	    // trigger kaxon horn: rising trigger of start
	    #RT_Start(CLK := #Start);
	    // trigger kaxon horn: rising trigger of stop
	    #RT_Stop(CLK := #Stop);
	    // trigger kaxon horn: rising trigger of fault
	    #RT_Fault(CLK := #GlobalFault);
	    // trigger kaxon horn: rising trigger of blockage
	    #RT_Blockage(CLK := #GlobalBlockage);
	    // trigger kaxon horn: rising trigger of estop
	    #RT_Estop(CLK := #EstopActive);
	    // trigger kaxon horn: rising trigger of fire
	    #RT_Fire(CLK := #Fire);
	    
	    // --------------
	    // Horn condition
	    // --------------
	    
	    #HornCondition :=
	    #RT_Start.Q OR
	    #RT_Stop.Q OR
	    #RT_Fire.Q OR
	    #RT_Fault.Q OR
	    #RT_Estop.Q OR
	    #RT_Fire.Q;
	    
	    // -------------------
	    // Horn alert duration
	    // -------------------
	    
	    #KlaxonHornTimer.TOF(IN := #HornCondition,
	                         PT := t#5s);
	    
	    #HornActive :=
	    #KlaxonHornTimer.Q;
	    
	END_REGION
	
	
	
	
	
	
	
	
	
	
	
	
	
END_FUNCTION_BLOCK
END_NAMESPACE

NAMESPACE ProductionLine
FUNCTION_BLOCK Flow_Test
{ S7_Optimized_Access := 'TRUE' ; Published := 'FALSE' }
VERSION : 0.1
   VAR 
      Start { S7_SetPoint := 'True'} : Bool;   //  // Start command (e.g. from I0.0)
      StartTest : Test_Logic;
      GoToRightDP1 : Test_Logic;
      ContinueStraightDP1 : Test_Logic;
      ContinueStraightDP2 : Test_Logic;
      GotorightDP2Thentoright : Test_Logic;
      GotorightDP2ThentoLeft : Test_Logic;
      ContinueStraightDP3 : Test_Logic;
      ContinueStraightDP4 : Test_Logic;
      GotoRightDP4 : Test_Logic;
      "A1.13.1_Straight" : Test_Logic;
      "A1.13.1_left" : Test_Logic;
      R_TRIG_Instance {InstructionName := 'R_TRIG'; LibVersion := '1.0'} : R_TRIG;
   END_VAR


BEGIN
	// ==========================================================================================================================================
	// Company        : LogTech, s.r.o.
	// Created by     : Mahmoud Elnady
	// Block          : FB_FlowTest
	// Project        : Lékárna Chrudim
	// Project number : 23-157
	// ==========================================================================================================================================
	
	REGION Start Test
	    #StartTest(Start := #Start,
	               StartPoint := _."A1.1.1",
	               EndPoint :=  _."A1.5.3");
	END_REGION
	
	
	REGION Go TO Right DP1
	    #GoToRightDP1(Start := DB_ToteTracking.Conveyor[_."A1.6.1"].ToteDir.toRight AND
	                  DB_ToteTracking.Conveyor[_."A1.6.2"].ToteDir.toRight AND
	                  _.ProductionLine.IDB_ProductionLine."A1.5.3".FilteredSensor,
	                  StartPoint := _."B1.1.1",
	                  EndPoint := _."B1.9.2");
	END_REGION
	
	
	REGION CONTINUE Straight DP1
	    
	    #ContinueStraightDP1(Start := DB_ToteTracking.Conveyor[_."A1.6.1"].ToteDir.Straight AND
	                         DB_ToteTracking.Conveyor[_."A1.6.2"].ToteDir.Straight AND
	                         _.ProductionLine.IDB_ProductionLine."A1.5.3".FilteredSensor,
	                         StartPoint := _."A1.7.1",
	                         EndPoint := _."A1.8.1");
	    
	END_REGION
	
	IF (DB_ToteTracking.Conveyor[_."A1.6.1"].ToteDir.Straight OR
	    DB_ToteTracking.Conveyor[_."A1.6.1"].ToteDir.toRight) AND
	    IDB_ProductionLine."A1.5.3".FilteredSensor
	THEN
	    _.Global.DB_SystemSimu.TriggerSensor.Line.ProductionLine.Conveyor[_."A1.6.1"] := TRUE;
	ELSE
	    _.Global.DB_SystemSimu.TriggerSensor.Line.ProductionLine.Conveyor[_."A1.6.1"] := FALSE;
	END_IF;
	
	
	        
	REGION CONTINUE Straight DP2
	    
	    #ContinueStraightDP2(Start := DB_ToteTracking.Conveyor[_."B1.10.1"].ToteDir.Straight AND
	                                  IDB_ProductionLine."B1.9.2".FilteredSensor,
	                         StartPoint := _."B1.11.1",
	                         EndPoint := _."B1.17.4");
	    
	END_REGION
	
	
	REGION Go TO Right DP2 THEN TO Right
	    #GotorightDP2Thentoright(Start := DB_ToteTracking.Conveyor[_."B1.10.1"].ToteDir.toRight AND
	                             DB_ToteTracking.Conveyor[_."C1.3.1"].ToteDir.toRight AND
	                             IDB_ProductionLine."B1.9.2".FilteredSensor,
	                             StartPoint := _."C1.2.2",
	                             EndPoint := _."C1.2.1");
	END_REGION
	
	
	REGION Go TO Right THEN TO Left
	    #GotorightDP2ThentoLeft(Start := DB_ToteTracking.Conveyor[_."B1.10.1"].ToteDir.toRight AND
	                            DB_ToteTracking.Conveyor[_."C1.3.1"].ToteDir.toLeft AND
	                            IDB_ProductionLine."B1.9.2".FilteredSensor,
	                            StartPoint := _."C1.4.1",
	                            EndPoint :=  _."C1.4.2");
	END_REGION
	
	
	IF (DB_ToteTracking.Conveyor[_."B1.10.1"].ToteDir.Straight OR
	    DB_ToteTracking.Conveyor[_."B1.10.1"].ToteDir.toRight) AND
	    IDB_ProductionLine."B1.9.2".FilteredSensor
	THEN
	    _.Global.DB_SystemSimu.TriggerSensor.Line.ProductionLine.Conveyor[_."B1.10.1"] := TRUE;
	ELSE
	    _.Global.DB_SystemSimu.TriggerSensor.Line.ProductionLine.Conveyor[_."B1.10.1"] := FALSE;
	END_IF;
	
	IF (DB_ToteTracking.Conveyor[_."C1.3.1"].ToteDir.toLeft OR
	    DB_ToteTracking.Conveyor[_."C1.3.1"].ToteDir.toRight) AND
	    IDB_ProductionLine."B1.10.1".FilteredSensor AND
	    DB_ToteTracking.Conveyor[_."B1.10.1"].ToteDir.toRight
	THEN
	    _.Global.DB_SystemSimu.TriggerSensor.Line.ProductionLine.Conveyor[_."C1.3.1"] := TRUE;
	ELSE
	    _.Global.DB_SystemSimu.TriggerSensor.Line.ProductionLine.Conveyor[_."C1.3.1"] := FALSE;
	END_IF;
	
	
	
	REGION CONTINUE Straight DP3
	    #ContinueStraightDP3(Start := DB_ToteTracking.Conveyor[_."B1.18.1"].ToteDir.Straight AND
	                                  IDB_ProductionLine."B1.17.4".FilteredSensor,
	                         StartPoint := _."B1.19.1",
	                         EndPoint := _."B1.23.1");
	END_REGION
	
	IF (DB_ToteTracking.Conveyor[_."B1.18.1"].ToteDir.toLeft OR
	    DB_ToteTracking.Conveyor[_."B1.18.1"].ToteDir.Straight) AND
	    IDB_ProductionLine."B1.17.4".FilteredSensor
	THEN
	    _.Global.DB_SystemSimu.TriggerSensor.Line.ProductionLine.Conveyor[_."B1.18.1"] := TRUE;
	ELSE
	    _.Global.DB_SystemSimu.TriggerSensor.Line.ProductionLine.Conveyor[_."B1.18.1"] := FALSE;
	END_IF;
	
	#R_TRIG_Instance(CLK:=( IDB_ProductionLine."B1.18.1".FilteredSensor AND
	                 DB_ToteTracking.Conveyor[_."B1.18.1"].ToteDir.toLeft));
	
	
	
	REGION CONTINUE Straight DP4
	    #ContinueStraightDP4(Start := DB_ToteTracking.Conveyor[_."A1.9.1"].ToteDir.Straight AND
	                         DB_ToteTracking.Conveyor[_."A1.9.2"].ToteDir.Straight AND
	                         _.ProductionLine.IDB_ProductionLine."A1.8.1".FilteredSensor,
	                         StartPoint := _."A1.10.1",
	                         EndPoint := _."A1.12.2");
	END_REGION
	
	
	REGION Go TO Right DP4
	    #GotoRightDP4(Start := DB_ToteTracking.Conveyor[_."A1.9.1"].ToteDir.toRight AND
	                  DB_ToteTracking.Conveyor[_."A1.9.2"].ToteDir.toRight AND
	                  _.ProductionLine.IDB_ProductionLine."A1.8.1".FilteredSensor,
	                  StartPoint := _."D1.1.1",
	                  EndPoint :=  _."D1.12.3");
	END_REGION
	
	IF (DB_ToteTracking.Conveyor[_."A1.9.1"].ToteDir.Straight OR
	    DB_ToteTracking.Conveyor[_."A1.9.1"].ToteDir.toRight) AND
	    IDB_ProductionLine."A1.8.1".FilteredSensor
	THEN
	    _.Global.DB_SystemSimu.TriggerSensor.Line.ProductionLine.Conveyor[_."A1.9.1"] := TRUE;
	ELSE
	    _.Global.DB_SystemSimu.TriggerSensor.Line.ProductionLine.Conveyor[_."A1.9.1"] := FALSE;
	END_IF;
	
	REGION A1.13.1_Straight
	    
	    #"A1.13.1_Straight"(Start:= DB_ToteTracking.Conveyor[_."A1.13.1"].ToteDir.Straight AND
	                                IDB_ProductionLine."A1.12.2".FilteredSensor,
	                        StartPoint:=_."A1.14.1",
	                        EndPoint:= _."A1.14.26");
	    
	   
	END_REGION
	        
	REGION A1.13.1_Left
	    
	    #"A1.13.1_left"(Start := DB_ToteTracking.Conveyor[_."A1.13.1"].ToteDir.toLeft AND
	                    IDB_ProductionLine."A1.12.2".FilteredSensor,
	                    StartPoint := _."A2.2.1",
	                    EndPoint := _."A2.2.26");
	    
	    
	END_REGION
	
	
	    
	    
	
END_FUNCTION_BLOCK
END_NAMESPACE

NAMESPACE ProductionLine
FUNCTION_BLOCK Test_Logic
{ S7_Optimized_Access := 'TRUE' ; Published := 'FALSE' }
VERSION : 0.1
   VAR_INPUT 
      Start : Bool;
      StartPoint : Int;
      EndPoint : Int;
   END_VAR

   VAR 
      Active : Bool;
      "Counter" : Int;
      PulseTimer {InstructionName := 'TON_TIME'; LibVersion := '1.0'; S7_SetPoint := 'False'} : TON_TIME;
   END_VAR


BEGIN
	// ==========================================================================================================================================
	// Company        : LogTech, s.r.o.
	// Created by     : Mahmoud Elnady
	// Block          : FB_LineA1
	// Project        : Lékárna Chrudim
	// Project number : 23-157
	// ==========================================================================================================================================
	
	REGION Start
	    // Start sequence
	    IF #Start AND NOT #Active THEN
	        #Active := TRUE;
	        #Counter := #StartPoint;               // Start from first output
	    END_IF;
	    
	    // Main pulse logic
	    IF #Active THEN
	        // Turn ON the current output
	        _.Global.DB_SystemSimu.TriggerSensor.Line.ProductionLine.Conveyor[#Counter] := TRUE;
	        #PulseTimer(IN := TRUE,
	                    PT := T#3s);
	        
	        // When timer expires
	        IF #PulseTimer.Q THEN
	            // Turn OFF current output
	            _.Global.DB_SystemSimu.TriggerSensor.Line.ProductionLine.Conveyor[#Counter] := FALSE;
	            
	            // Reset timer
	            RESET_TIMER(#PulseTimer);
	            
	            // Move to next output
	            #Counter := #Counter + 1;
	            
	            // Stop if last output finished
	            IF #Counter > #EndPoint THEN
	                #Active := FALSE;
	            END_IF;
	        END_IF;
	    ELSE
	        // Make sure all outputs are OFF when not active
	        (* FOR #var_i := 1001 TO #N DO
	        //#Q[#var_i] := FALSE;
	        _.Global.DB_SystemSimu.TriggerSensor.Line.ProductionLine.Conveyor[#Counter] := FALSE;
	    END_FOR;*)
	        RESET_TIMER(#PulseTimer);
	    END_IF;
	END_REGION
END_FUNCTION_BLOCK
END_NAMESPACE

NAMESPACE ProductionLine
FUNCTION_BLOCK BarcodeReader
{ S7_Optimized_Access := 'TRUE' ; Published := 'FALSE' }
VERSION : 0.1
   VAR 
      DP1 { S7_SetPoint := 'False'} : _.Global.DataMan262;
      DP2 { S7_SetPoint := 'False'} : _.Global.DataMan262;
      DP3 { S7_SetPoint := 'False'} : _.Global.DataMan262;
      DP4 { S7_SetPoint := 'False'} : _.Global.DataMan262;
   END_VAR


BEGIN
	// ==========================================================================================================================================
	// Company        : LogTech, s.r.o.
	// Created by     : Mahmoud Elnady
	// Block          : Barcode Reader
	// Project        : Lekarna, Chrudim -PLC001 -MCC001
	// Project number : 23-157
	// ==========================================================================================================================================
	
	REGION DP1
	    
	    #DP1(TriggerSignal:= IDB_ProductionLine."A1.5.1".FilteredSensor,
	         "Dataman-Results Available":=_."DP1-Results Available",
	         "Dataman-TriggerReady":=_."DP1-TriggerReady",
	         "Dataman-TriggerAck":=_."DP1-TriggerAck",
	         "Dataman-ResultID":=_."DP1-ResultID",
	         "Dataman-Result Code":=_."DP1-Result Code",
	         "Dataman-Result Length":=_."DP1-Result Length",
	         "Result Data":=_."Result data_DP1",
	         "Dataman-UserData Length"=>_."DP1-UserData Length",
	         "Dataman-UserData Option"=>_."DP1-UserData Option",
	         "User Data"=>_.UserData_DP1,
	         "Dataman-TriggerEnable":=_."DP1-TriggerEnable",
	         "Dataman-Trigger":=_."DP1-Trigger",
	         "Dataman-ResultsAck":=_."DP1-ResultsAck");
	    
	END_REGION
	
	REGION DP2
	    
	    #DP2(TriggerSignal := IDB_ProductionLine."B1.9.1".FilteredSensor,
	         "Dataman-Results Available" := _."DP2-Results Available",
	         "Dataman-TriggerReady" := _."DP2-TriggerReady",
	         "Dataman-TriggerAck" := _."DP2-TriggerAck",
	         "Dataman-ResultID" := _."DP2-ResultID",
	         "Dataman-Result Code" := _."DP2-Result Code",
	         "Dataman-Result Length" := _."DP2-Result Length",
	         "Result Data" := _."Result data_DP2",
	         "Dataman-UserData Length" => _."DP2-UserData Length",
	         "Dataman-UserData Option" => _."DP2-UserData Option",
	         "User Data" => _.UserData_DP2,
	         "Dataman-TriggerEnable" := _."DP2-TriggerEnable",
	         "Dataman-Trigger" := _."DP2-Trigger",
	         "Dataman-ResultsAck" := _."DP2-ResultsAck");
	    
	END_REGION
	
	REGION DP3
	    
	    #DP3(TriggerSignal := IDB_ProductionLine."B1.17.1".FilteredSensor,
	         "Dataman-Results Available" := _."DP3-Results Available",
	         "Dataman-TriggerReady" := _."DP3-TriggerReady",
	         "Dataman-TriggerAck" := _."DP3-TriggerAck",
	         "Dataman-ResultID" := _."DP3-ResultID",
	         "Dataman-Result Code" := _."DP3-Result Code",
	         "Dataman-Result Length" := _."DP3-Result Length",
	         "Result Data" := _."Result data_DP3",
	         "Dataman-UserData Length" => _."DP3-UserData Length",
	         "Dataman-UserData Option" => _."DP3-UserData Option",
	         "User Data" => _.UserData_DP3,
	         "Dataman-TriggerEnable" := _."DP3-TriggerEnable",
	         "Dataman-Trigger" := _."DP3-Trigger",
	         "Dataman-ResultsAck" := _."DP3-ResultsAck");
	    
	END_REGION
	
	
	REGION DP4
	    
	    #DP4(TriggerSignal := IDB_ProductionLine."A1.7.4".FilteredSensor,
	         "Dataman-Results Available" := _."DP4-Results Available",
	         "Dataman-TriggerReady" := _."DP4-TriggerReady",
	         "Dataman-TriggerAck" := _."DP4-TriggerAck",
	         "Dataman-ResultID" := _."DP4-ResultID",
	         "Dataman-Result Code" := _."DP4-Result Code",
	         "Dataman-Result Length" := _."DP4-Result Length",
	         "Result Data" := _."Result data_DP4",
	         "Dataman-UserData Length" => _."DP4-UserData Length",
	         "Dataman-UserData Option" => _."DP4-UserData Option",
	         "User Data" => _.UserData_DP4,
	         "Dataman-TriggerEnable" := _."DP4-TriggerEnable",
	         "Dataman-Trigger" := _."DP4-Trigger",
	         "Dataman-ResultsAck" := _."DP4-ResultsAck");
	    
	END_REGION
	
END_FUNCTION_BLOCK
END_NAMESPACE

NAMESPACE ProductionLine
FUNCTION_BLOCK FB_OPC_Communication
{ S7_Optimized_Access := 'TRUE' ; Published := 'FALSE' }
VERSION : 0.1
   VAR 
      Communication_DP1 { S7_SetPoint := 'False'} : FB_OPC_DestRequest;
      Communication_DP2 { S7_SetPoint := 'False'} : FB_OPC_DestRequest;
      Communication_DP3 { S7_SetPoint := 'False'} : FB_OPC_DestRequest;
      Communication_DP4 { S7_SetPoint := 'False'} : FB_OPC_DestRequest;
      Communication_IP1 { S7_SetPoint := 'False'} : FB_OPC_DestInfo;
      Communication_IP2 { S7_SetPoint := 'False'} : FB_OPC_DestInfo;
      Communication_IP3 { S7_SetPoint := 'False'} : FB_OPC_DestInfo;
      Communication_IP4 { S7_SetPoint := 'False'} : FB_OPC_DestInfo;
      Communication_IP5 { S7_SetPoint := 'False'} : FB_OPC_DestInfo;
      Communication_IP6 { S7_SetPoint := 'False'} : FB_OPC_DestInfo;
      Communication_IP7 { S7_SetPoint := 'False'} : FB_OPC_DestInfo;
      Communication_IP8 { S7_SetPoint := 'False'} : FB_OPC_DestInfo;
      Communication_IP9 { S7_SetPoint := 'False'} : FB_OPC_DestInfo;
      Communication_SYS_OP { S7_SetPoint := 'False'} : FB_OPC_SysStatus;
      Communication_SYS_OP_Source : OPC_SystemStatus;
      Communication_SYS_OP_Ack : OPC_SystStatus_Ack;
      timPeriodicSend {InstructionName := 'IEC_TIMER'; LibVersion := '1.0'} : IEC_TIMER;
      timWatchdog {InstructionName := 'IEC_TIMER'; LibVersion := '1.0'} : IEC_TIMER;
      Communication_fault : Bool;
   END_VAR


BEGIN
	// ==========================================================================================================================================
	// Company        : LogTech, s.r.o.
	// Created by     : Mahmoud Elnady
	// Block          : FB_OPC_Communication
	// Project        : Lekarna, Chrudim -PLC001 -MCC001
	// Project number : 23-157
	// ==========================================================================================================================================
	
	//------------------------------------------------------
	// Initialization
	//------------------------------------------------------
	
	REGION Initialization
	    // Initialization section to reset the sequence numbers at the first scan
	    IF _.DB_Sync.memoryBit.FirstScan THEN
	        OPC_Data.DP1.DestRequest.Source.SourceSeq := 0;
	        OPC_Data.DP2.DestRequest.Source.SourceSeq := 0;
	        OPC_Data.DP3.DestRequest.Source.SourceSeq := 0;
	        OPC_Data.DP4.DestRequest.Source.SourceSeq := 0;
	        OPC_Data.IP11.DestInfo.Source.SourceSeq := 0;
	        OPC_Data.IP12.DestInfo.Source.SourceSeq := 0;
	        OPC_Data.IP21.DestInfo.Source.SourceSeq := 0;
	        OPC_Data.IP22.DestInfo.Source.SourceSeq := 0;
	        OPC_Data.IP23.DestInfo.Source.SourceSeq := 0;
	        OPC_Data.IP31.DestInfo.Source.SourceSeq := 0;
	        OPC_Data.IP32.DestInfo.Source.SourceSeq := 0;
	        OPC_Data.IP41.DestInfo.Source.SourceSeq := 0;
	        OPC_Data.IP42.DestInfo.Source.SourceSeq := 0;
	    END_IF;
	END_REGION
	
	//------------------------------------------------------
	// Handle destination request/ destination Information communication
	//------------------------------------------------------
	
	REGION DP1- DestRequest
	    // Handle destination request communication for DP1
	    #Communication_DP1(Source := OPC_Data.DP1.DestRequest.Source,
	                       Ack := OPC_Data.DP1.DestRequest.Ack);
	    
	END_REGION
	
	
	REGION DP2- DestRequest
	    // Handle destination request communication for DP2
	    #Communication_DP2(Source := OPC_Data.DP2.DestRequest.Source,
	                       Ack := OPC_Data.DP2.DestRequest.Ack);
	END_REGION
	
	
	REGION DP3- DestRequest
	    // Handle destination request communication for DP3
	    #Communication_DP3(Source := OPC_Data.DP3.DestRequest.Source,
	                       Ack := OPC_Data.DP3.DestRequest.Ack);
	END_REGION
	
	
	REGION DP4- DestRequest
	    // Handle destination request communication for DP4
	    #Communication_DP4(Source := OPC_Data.DP4.DestRequest.Source,
	                       Ack := OPC_Data.DP4.DestRequest.Ack);
	END_REGION
	
	REGION DS1- DestRequest
	    // Handle destination information communication for DS1
	    #Communication_IP1(Source := OPC_Data.IP11.DestInfo.Source,
	                       Ack := OPC_Data.IP11.DestInfo.Ack);
	END_REGION
	
	
	REGION DS2- DestRequest
	    // Handle destination information communication for DS2
	    #Communication_IP2(Source := OPC_Data.IP12.DestInfo.Source,
	                       Ack := OPC_Data.IP12.DestInfo.Ack);
	END_REGION
	
	
	REGION DS3- DestRequest
	    // Handle destination information communication for DS3
	    #Communication_IP3(Source := OPC_Data.IP21.DestInfo.Source,
	                       Ack := OPC_Data.IP21.DestInfo.Ack);
	END_REGION
	
	
	REGION DS4- DestRequest
	    // Handle destination information communication for DS4
	    #Communication_IP4(Source := OPC_Data.IP22.DestInfo.Source,
	                       Ack := OPC_Data.IP22.DestInfo.Ack);
	END_REGION
	
	REGION DS5- DestRequest
	    // Handle destination information communication for DS4
	    #Communication_IP5(Source := OPC_Data.IP23.DestInfo.Source,
	                       Ack := OPC_Data.IP23.DestInfo.Ack);
	END_REGION
	
	REGION DS6- DestRequest
	    // Handle destination information communication for DS4
	    #Communication_IP6(Source := OPC_Data.IP31.DestInfo.Source,
	                       Ack := OPC_Data.IP31.DestInfo.Ack);
	END_REGION
	
	REGION DS7- DestRequest
	    // Handle destination information communication for DS4
	    #Communication_IP7(Source := OPC_Data.IP32.DestInfo.Source,
	                       Ack := OPC_Data.IP32.DestInfo.Ack);
	END_REGION
	
	REGION DS8- DestRequest
	    // Handle destination information communication for DS4
	    #Communication_IP8(Source := OPC_Data.IP41.DestInfo.Source,
	                       Ack := OPC_Data.IP41.DestInfo.Ack);
	END_REGION
	
	REGION DS9- DestRequest
	    // Handle destination information communication for DS4
	    #Communication_IP9(Source := OPC_Data.IP42.DestInfo.Source,
	                       Ack := OPC_Data.IP42.DestInfo.Ack);
	END_REGION
	
	//------------------------------------------------------
	//Handle communication for overall system operation status
	//------------------------------------------------------
	
	REGION  SystStatus
	    // Statement section REGION
	    #Communication_SYS_OP(Source:=#Communication_SYS_OP_Source,
	                          Ack:=#Communication_SYS_OP_Ack);
	    
	END_REGION
	
	
	//------------------------------------------------------
	// Heart Beats
	//------------------------------------------------------
	
	REGION SYS Position - SystStatus
	    // // Periodic communication trigger for system status data (SYS_OP)
	    IF NOT #timPeriodicSend.Q THEN
	        #Communication_SYS_OP.Comm.Send := TRUE;
	    END_IF;
	    
	    #timPeriodicSend.TON(IN := #Communication_SYS_OP.Comm.Send AND
	                               #Communication_SYS_OP.Comm.Send_prev,
	                         PT := T#10s);
	    IF #timPeriodicSend.Q THEN
	        #Communication_SYS_OP.Comm.Send := FALSE;
	    END_IF;
	    
	    
	END_REGION
	
	//Periodic Counter, incremented every 10 seconds.
	//IF one side does NOT increment the counter within 30 seconds,
	//it will be considered offline BY the other side.
	REGION Watchdog
	    
	    OPC_Data.Watchdog.Keep_Alive_PLC := #Communication_SYS_OP.Comm.SourceSeq;
	    
	    #Communication_SYS_OP.Comm.AckSeq := OPC_Data.Watchdog.Keep_Alive_WMS;
	    
	END_REGION
	
	
	REGION Communication Fault
	    
	    #timWatchdog.TON(IN :=  #Communication_SYS_OP.Comm.SourceSeq <> #Communication_SYS_OP.Comm.AckSeq ,
	                          PT := T#30s);
	    
	    IF #timWatchdog.Q THEN
	        #Communication_fault := TRUE;
	    ELSE
	        #Communication_fault := FALSE;
	    END_IF;
	    
	    //Global status
	    _.Global.DB_VisuColor.Line.ProductionLine.OPC.%X0 :=NOT #Communication_fault;
	    
	END_REGION
	
	//------------------------------------------------------
	// Status of Segment for WMS
	//------------------------------------------------------
	
	REGION Status OF Segment FOR WMS
	    // Status of Segment for WMS
	    //Update system status based on Flow Rack Loop status
	    IF IDB_Segments_Status.FlowRackLoopReadyToRun THEN
	        // If conveyor is ready, set OPC system status to '1'
	        OPC_Data.Status.Segment.FlowRackLoop := 1;
	    ELSE
	        // If not ready, set system status to '0'
	        OPC_Data.Status.Segment.FlowRackLoop := 0;
	    END_IF;
	    
	    IF IDB_Segments_Status.FlowRackWorkPlaceRightReadyToRun THEN
	        OPC_Data.Status.Segment.FlowRackWorkplaceRight := 1;
	    ELSE
	        OPC_Data.Status.Segment.FlowRackWorkplaceRight := 0;
	    END_IF;
	    
	    IF IDB_Segments_Status.FlowRackWorkPlaceLeftReadyToRun THEN
	        OPC_Data.Status.Segment.FlowRackWorkplaceLeft := 1;
	    ELSE
	        OPC_Data.Status.Segment.FlowRackWorkplaceLeft := 0;
	    END_IF;
	    
	    IF IDB_Segments_Status.FragileloopReadyToRun THEN
	        OPC_Data.Status.Segment.FragileLoop := 1;
	    ELSE
	        OPC_Data.Status.Segment.FragileLoop := 0;
	    END_IF;
	    
	END_REGION
	
	
	
	
	
	
	
	
	
	
	
	
END_FUNCTION_BLOCK
END_NAMESPACE

NAMESPACE ProductionLine
FUNCTION_BLOCK FB_OPC_DestAssigne
{ S7_Optimized_Access := 'TRUE' ; Published := 'FALSE' }
VERSION : 0.1
   VAR_IN_OUT 
      Source : OPC_DestAssign;
      Ack : OPC_DestAssign_Ack;
   END_VAR

   VAR 
      Communication { S7_SetPoint := 'False'} : FB_OPC_ReceiveSendAck;
      staSource : OPC_DestAssign;
      staAck : OPC_DestAssign_Ack;
   END_VAR

   VAR_TEMP 
      Retval : Int;
   END_VAR


BEGIN
	// ==========================================================================================================================================
	// Company        : LogTech, s.r.o.
	// Created by     : Mahmoud Elnady
	// Block          : OPC_SendReciveAck
	// Project        : Lekarna, Chrudim -PLC001 -MCC001
	// Project number : 23-157
	// ==========================================================================================================================================
	
	//======================================================
	// Region: Communication Handling and Logging
	// Description: Manages the communication routine and logs
	//              events for message sending, acknowledgment
	//              reception, and acknowledgment timeout.
	//======================================================
	
	//------------------------------------------------------
	// Call communication routine
	//------------------------------------------------------
	
	REGION Communication routine
	    // Call communication routine
	    #Communication(SourceSeq := #staSource.SourceSeq,
	                   AckSeq := #staAck.AckSeq);
	END_REGION
	
	#Source.SourceSeq := #staSource.SourceSeq;
	#staAck.AckSeq := #Ack.AckSeq;
	
	
	//------------------------------------------------------
	// Log event when a new message is sent
	//------------------------------------------------------
	
	REGION Log event - new message
	    IF #Communication.Log.New_data_received THEN
	        #Communication.Log.New_data_received := FALSE;
	        // Logging
	        //(LOG)3005=$ Node $, new message received, seq: $, palletID: $, WMSID $, destination: $, no-stretch: $
	        DB_LogMsg.LogMsg_9.Para_STRING_01.Data := #Source.SourceNode;
	        DB_LogMsg.LogMsg_9.Para_BYTE_02.Data := #Source.SourceSeq;
	        DB_LogMsg.LogMsg_9.Para_STRING_03.Data := #Source.TotesID;
	        DB_LogMsg.LogMsg_9.Para_STRING_04.Data := #Source.WMSID;
	        DB_LogMsg.LogMsg_9.Para_STRING_05.Data := #Source.DestinationNode;
	        #Retval := FC_LogMsg(EventID := 3005, EventLevel := 2, EventGroup := 33, LogMsg := DB_LogMsg.LogMsg_9);
	    END_IF;
	END_REGION
	
	//------------------------------------------------------
	// Log event when new acknowledgment is received
	//------------------------------------------------------
	
	REGION Log event-New acknowledgment
	    IF #Communication.Log.Ack_send THEN
	        #Communication.Log.Ack_send := FALSE;
	        // Logging
	        //(LOG)3006=$ Node $, acknowledge sent, seq: $, palletID: $, WMSID: $, confirmation: $
	        DB_LogMsg.LogMsg_10.Para_STRING_01.Data := #Ack.SourceNode;
	        DB_LogMsg.LogMsg_10.Para_BYTE_02.Data := #Ack.AckSeq;
	        DB_LogMsg.LogMsg_10.Para_STRING_03.Data := #Ack.TotesID;
	        DB_LogMsg.LogMsg_10.Para_STRING_04.Data := #Ack.WMSID;
	        DB_LogMsg.LogMsg_10.Para_CHAR_05.Data := STRING_TO_CHAR(#Ack.Confirmation);
	        #Retval := FC_LogMsg(EventID := 3006, EventLevel := 2, EventGroup := 33, LogMsg := DB_LogMsg.LogMsg_10);
	    END_IF;
	END_REGION
	
	
END_FUNCTION_BLOCK
END_NAMESPACE

NAMESPACE ProductionLine
FUNCTION_BLOCK FB_OPC_DestInfo
{ S7_Optimized_Access := 'TRUE' ; Published := 'FALSE' }
VERSION : 0.1
   VAR_IN_OUT 
      Source : OPC_DestInfo;
      Ack : OPC_DestInfo_Ack;
   END_VAR

   VAR 
      Communication { S7_SetPoint := 'False'} : FB_OPC_SendReciveAck;
      staSource { ExternalAccessible := 'False'; ExternalVisible := 'False'; ExternalWritable := 'False'; S7_SetPoint := 'False'} : OPC_DestInfo;
      staAck { ExternalAccessible := 'False'; ExternalVisible := 'False'; ExternalWritable := 'False'; S7_SetPoint := 'False'} : OPC_DestInfo_Ack;
   END_VAR

   VAR_TEMP 
      Retval : Int;
   END_VAR


BEGIN
	// ==========================================================================================================================================
	// Company        : LogTech, s.r.o.
	// Created by     : Mahmoud Elnady
	// Block          : OPC_SendReciveAck
	// Project        : Lekarna, Chrudim -PLC001 -MCC001
	// Project number : 23-157
	// ==========================================================================================================================================
	
	
	//======================================================
	// Region: Communication Handling and Logging
	// Description: Manages the communication routine and logs
	//              events for message sending, acknowledgment
	//              reception, and acknowledgment timeout.
	//======================================================
	
	//------------------------------------------------------
	// Call communication routine
	//------------------------------------------------------
	REGION Communication routine
	    // Call communication routine
	    #Communication(SourceSeq := #staSource.SourceSeq,
	                   AckSeq := #staAck.AckSeq,
	                   Timeout := T#20s);
	END_REGION
	
	#Source.SourceSeq := #staSource.SourceSeq;
	#staAck.AckSeq := #Ack.AckSeq;
	
	
	//------------------------------------------------------
	// Log event when a new message is sent
	//------------------------------------------------------
	
	REGION Log event - new message
	    IF #Communication.Log.Send THEN
	        #Communication.Log.Send := FALSE;
	        // Logging
	        //(LOG)3003=$ Node $, new message sent, seq: $, palletID: $, WMSID: $
	        DB_LogMsg.LogMsg_7.Para_STRING_01.Data := #Source.DecisionPoint;
	        DB_LogMsg.LogMsg_7.Para_BYTE_02.Data := #Source.SourceSeq;
	        DB_LogMsg.LogMsg_7.Para_STRING_03.Data := #Source.Barcode;
	        DB_LogMsg.LogMsg_7.Para_STRING_04.Data := #Source.InformationPoint;
	        #Retval := FC_LogMsg(EventID := 3003, EventLevel := 2, EventGroup := 33, LogMsg := DB_LogMsg.LogMsg_7);
	    END_IF;
	END_REGION
	
	//------------------------------------------------------
	// Log event when new acknowledgment is received
	//------------------------------------------------------
	
	REGION Log event-New acknowledgment
	    IF #Communication.Log.New_Ack_received THEN
	        #Communication.Log.New_Ack_received := FALSE;
	        // Logging
	        //(LOG)3004=$ Node $, acknowledge received, seq: $, palletID: $, WMSID: $
	        DB_LogMsg.LogMsg_7.Para_BYTE_02.Data := #Ack.AckSeq;
	        #Retval := FC_LogMsg(EventID := 3004, EventLevel := 2, EventGroup := 33, LogMsg := DB_LogMsg.LogMsg_7);
	    END_IF;
	END_REGION
	
	//------------------------------------------------------
	// Log event when acknowledgment timeout occurs
	//------------------------------------------------------
	
	REGION Log event- acknowledgment timeout
	    IF #Communication.Log.Ack_timeout THEN
	        #Communication.Log.Ack_timeout := FALSE;
	        // Logging
	        //(LOG)3009=$ Node $, seq: $, acknowledge timeout!
	        DB_LogMsg.LogMsg_8.Para_STRING_01.Data := #Source.DecisionPoint;
	        DB_LogMsg.LogMsg_8.Para_BYTE_02.Data := #Communication.SendSeq;
	        #Retval := FC_LogMsg(EventID := 3009, EventLevel := 3, EventGroup := 33, LogMsg := DB_LogMsg.LogMsg_8);
	    END_IF;
	END_REGION
	
END_FUNCTION_BLOCK
END_NAMESPACE

NAMESPACE ProductionLine
FUNCTION_BLOCK FB_OPC_DestRequest
{ S7_Optimized_Access := 'TRUE' ; Published := 'FALSE' }
VERSION : 0.1
   VAR_IN_OUT 
      Source : OPC_DsetRequest;
      Ack : OPC_DestRequest_Ack;
   END_VAR

   VAR 
      Communication { S7_SetPoint := 'False'} : FB_OPC_SendReciveAck;
      staSource { ExternalAccessible := 'False'; ExternalVisible := 'False'; ExternalWritable := 'False'; S7_SetPoint := 'False'} : OPC_DsetRequest;
      staAck { ExternalAccessible := 'False'; ExternalVisible := 'False'; ExternalWritable := 'False'; S7_SetPoint := 'False'} : OPC_DestRequest_Ack;
   END_VAR

   VAR_TEMP 
      Retval : Int;
   END_VAR


BEGIN
	// ==========================================================================================================================================
	// Company        : LogTech, s.r.o.
	// Created by     : Mahmoud Elnady
	// Block          : OPC_SendReciveAck
	// Project        : Lekarna, Chrudim -PLC001 -MCC001
	// Project number : 23-157
	// ==========================================================================================================================================
	
	//======================================================
	// Region: Communication Handling and Logging
	// Description: Manages the communication routine and logs
	//              events for message sending, acknowledgment
	//              reception, and acknowledgment timeout.
	//======================================================
	
	//------------------------------------------------------
	// Call communication routine
	//------------------------------------------------------
	 REGION Communication Routine
	    // Call communication routine
	    #Communication(Timeout := T#15s,
	                   SourceSeq := #staSource.SourceSeq,
	                   AckSeq := #staAck.AckSeq);
	END_REGION 
	
	#Source.SourceSeq := #staSource.SourceSeq;
	#staAck.AckSeq := #Ack.AckSeq;
	
	//------------------------------------------------------
	// Log event when a new message is sent
	//------------------------------------------------------
	
	REGION Log event - new message
	    IF #Communication.Log.Send THEN
	        #Communication.Log.Send := FALSE;
	        // Logging
	        //(LOG)3001=$ Node $, new message sent, seq: $, palletID: $, WMSID $, barcode: $, weight: $, height: $, width: $, length: $, quality: $
	        DB_LogMsg.LogMsg_4.Para_STRING_01.Data := #Source.DecisionPoint;
	        DB_LogMsg.LogMsg_4.Para_BYTE_02.Data := #Source.SourceSeq;
	        //"DB_LogMsg".LogMsg_4.Para_STRING_03.Data := #Source.TotesID;
	        //"DB_LogMsg".LogMsg_4.Para_STRING_04.Data := #Source.WMSID;
	        DB_LogMsg.LogMsg_4.Para_STRING_05.Data := #Source.Barcode;
	        //"DB_LogMsg".LogMsg_4.Para_STRING_06.Data := #Source.Weight;
	               //"DB_LogMsg".LogMsg_4.Para_CHAR_09.Data := STRING_TO_CHAR(#Source.Length);
	        //"DB_LogMsg".LogMsg_4.Para_CHAR_10.Data := STRING_TO_CHAR(#Source.Quality);
	        
	        #Retval := FC_LogMsg(EventID := 3001,
	                               EventLevel := 2,
	                               EventGroup := 33,
	                               LogMsg := DB_LogMsg.LogMsg_4);
	    END_IF;
	END_REGION
	
	//------------------------------------------------------
	// Log event when new acknowledgment is received
	//------------------------------------------------------
	
	REGION Log event-New acknowledgment
	    IF #Communication.Log.New_Ack_received THEN
	        #Communication.Log.New_Ack_received := FALSE;
	        // Logging
	        //(LOG)3002=$ Node $, acknowledge received, seq: $, palletID: $, WMSID $, destination: $, no-stretch: $
	        DB_LogMsg.LogMsg_5.Para_STRING_01.Data := #Ack.DecisionPoint;
	        DB_LogMsg.LogMsg_5.Para_BYTE_02.Data := #Ack.AckSeq;
	        DB_LogMsg.LogMsg_5.Para_STRING_03.Data := #Ack.Barcode;
	        //"DB_LogMsg".LogMsg_5.Para_STRING_04.Data := #Ack.WMSID;
	        DB_LogMsg.LogMsg_5.Para_STRING_05.Data := #Ack.Destination;
	        
	        #Retval := FC_LogMsg(EventID := 3002,
	                               EventLevel := 2,
	                               EventGroup := 33,
	                               LogMsg := DB_LogMsg.LogMsg_5);
	    END_IF;
	END_REGION
	
	//------------------------------------------------------
	// Log event when acknowledgment timeout occurs
	//------------------------------------------------------
	
	REGION Log event- acknowledgment timeout
	    IF #Communication.Log.Ack_timeout THEN
	        #Communication.Log.Ack_timeout := FALSE;
	        // Logging
	        //(LOG)3009=$ Node $, seq: $, acknowledge timeout!
	        DB_LogMsg.LogMsg_6.Para_STRING_01.Data := #Source.DecisionPoint;
	        DB_LogMsg.LogMsg_6.Para_BYTE_02.Data := #Communication.SendSeq;
	        #Retval := FC_LogMsg(EventID := 3009,
	                               EventLevel := 3,
	                               EventGroup := 33,
	                               LogMsg := DB_LogMsg.LogMsg_6);
	    END_IF;
	END_REGION
	
	
	
END_FUNCTION_BLOCK
END_NAMESPACE

NAMESPACE ProductionLine
FUNCTION_BLOCK FB_OPC_ReceiveSendAck
{ S7_Optimized_Access := 'TRUE' ; Published := 'FALSE' }
VERSION : 0.1
   VAR_IN_OUT 
      SourceSeq : Int;
      AckSeq : Int;
   END_VAR

   VAR 
      New_data_received : Bool;
      Ack_send : Bool;
      Log : Struct
         New_data_received : Bool;
         Ack_send : Bool;
      END_STRUCT;
   END_VAR


BEGIN
	// ==========================================================================================================================================
	// Company        : LogTech, s.r.o.
	// Created by     : Mahmoud Elnady
	// Block          : OPC_SendReciveAck
	// Project        : Lekarna, Chrudim -PLC001 -MCC001
	// Project number : 23-157
	// ==========================================================================================================================================
	
	// =========================
	// REGION: Acknowledgement Handling
	// =========================
	// This region handles sending an acknowledgment signal.
	// When #Ack_send is TRUE, it means an ACK needs to be sent for the last received sequence.
	// The ACK sequence is set equal to the source sequence to confirm receipt.
	// Then, #Ack_send is reset to FALSE, and a log flag is set to indicate ACK was sent.
	
	REGION Ack_Handling
	    
	    IF #Ack_send THEN
	        #AckSeq := #SourceSeq;        // Update ACK sequence to match source sequence
	        #Ack_send := FALSE;           // Reset ACK send request
	        #Log.Ack_send := TRUE;        // Set log flag for diagnostics or monitoring
	    END_IF;
	    
	END_REGION
	
	
	// =========================
	// REGION: New Data Detection
	// =========================
	// This region checks if a new data sequence has been received.
	// If the source and ACK sequences are not equal, it determines if it's truly new data:
	// - If both sequences are non-zero, or source is 1 and ACK is 0 (initial start case),
	//   then new data is considered received.
	// - Otherwise, it assumes the ACK was missed and sets ACK to current source.
	
	REGION New_Data_Detection
	    
	    IF #SourceSeq <> #AckSeq THEN
	        // Check if both sequences are valid (non-zero), or it's the initial case (1,0)
	        IF (#SourceSeq <> 0 AND #AckSeq <> 0) OR (#SourceSeq = 1 AND #AckSeq = 0) THEN
	            #New_data_received := TRUE;           // Flag new data received
	            #Log.#New_data_received := TRUE;      // Set log flag for diagnostics
	        ELSE
	            #AckSeq := #SourceSeq;                // Treat as missed ACK and sync
	        END_IF;
	    END_IF;
	    
	END_REGION
	
END_FUNCTION_BLOCK
END_NAMESPACE

NAMESPACE ProductionLine
FUNCTION_BLOCK FB_OPC_SendReciveAck
{ S7_Optimized_Access := 'TRUE' ; Published := 'FALSE' }
VERSION : 0.1
   VAR_INPUT 
      Timeout : Time;
   END_VAR

   VAR_IN_OUT 
      SourceSeq : Int;
      AckSeq : Int;
   END_VAR

   VAR 
      Send : Bool;
      New_Ack_received : Bool;
      Ack_timeout : Bool;
      Send_prev : Bool;
      SendSeq : Int;
      TimeoutTimmer {InstructionName := 'IEC_TIMER'; LibVersion := '1.0'; S7_SetPoint := 'False'} : IEC_TIMER;
      Log : Struct
         Send : Bool;
         New_Ack_received : Bool;
         Ack_timeout : Bool;
      END_STRUCT;
   END_VAR

   VAR CONSTANT 
      maxInc : Int := 9999;
   END_VAR


BEGIN
	// ==========================================================================================================================================
	// Company        : LogTech, s.r.o.
	// Created by     : Mahmoud Elnady
	// Block          : OPC_SendReciveAck
	// Project        : Lekarna, Chrudim -PLC001 -MCC001
	// Project number : 23-157
	// ==========================================================================================================================================
	
	// REGION: Handle New Send Request
	REGION Handle_Send_Request
	    // Triggered on rising edge of #Send signal
	    IF #Send AND NOT #Send_prev THEN
	         #AckSeq := 0;  // Reset acknowledgment sequence
	        
	        // Increment source sequence, wrapping around after 99999 (B#16#270F)
	         IF #SourceSeq <> #maxInc THEN
	             #SourceSeq += 1;
	         ELSE
	             #SourceSeq := 1;
	         END_IF;
	        
	        #SendSeq := #SourceSeq;       // Set current send sequence
	        #New_Ack_received := FALSE;   // Reset acknowledgment flag
	        #Log.Send := TRUE;            // Log send event
	    END_IF;
	END_REGION
	
	// REGION: Process Acknowledgment
	REGION Process_Acknowledgment
	    IF #Send THEN
	        // Check if acknowledgment is received for the current send
	        IF #AckSeq = #SendSeq THEN
	            IF #AckSeq <> 0 THEN
	                #New_Ack_received := TRUE;     // Mark new acknowledgment
	                #Ack_timeout := FALSE;         // Clear timeout flag
	                #Log.#New_Ack_received := TRUE; // Log acknowledgment
	            END_IF;
	            //#Send := FALSE;  // Reset send signal
	        END_IF;
	    END_IF;
	    
	    // Update previous send state
	    #Send_prev := #Send;
	END_REGION
	
	
	// REGION: Timeout Management and Retransmission
	REGION Handle_Send_Timeout
	    // Activate timeout timer if timeout value is set
	    IF #Timeout <> T#0s THEN
	        #TimeoutTimmer.TON(IN := #Send AND NOT #New_Ack_received ,
	                           PT := #Timeout);
	    END_IF;
	    
	    // On timeout expiration, trigger retransmission logic
	    IF #TimeoutTimmer.Q THEN
	        #Send_prev := FALSE;         // Reset previous send to retrigger
	        #Ack_timeout := TRUE;        // Mark acknowledgment timeout
	        #Log.Ack_timeout := TRUE;    // Log timeout event
	        RESET_TIMER(#TimeoutTimmer); // Reset timer
	    END_IF;
	END_REGION
	
	
	
	
END_FUNCTION_BLOCK
END_NAMESPACE

NAMESPACE ProductionLine
FUNCTION_BLOCK FB_OPC_SysStatus
{ S7_Optimized_Access := 'TRUE' ; Published := 'FALSE' }
VERSION : 0.1
   VAR_IN_OUT 
      Source : OPC_SystemStatus;
      Ack : OPC_SystStatus_Ack;
   END_VAR

   VAR 
      Comm { S7_SetPoint := 'False'} : FB_OPC_SendReciveAck;
      staSource { ExternalAccessible := 'False'; ExternalVisible := 'False'; ExternalWritable := 'False'; S7_SetPoint := 'False'} : OPC_SystemStatus;
      staAck { ExternalAccessible := 'False'; ExternalVisible := 'False'; ExternalWritable := 'False'; S7_SetPoint := 'False'} : OPC_SystStatus_Ack;
   END_VAR

   VAR_TEMP 
      Retval : Int;
   END_VAR


BEGIN
	// ==========================================================================================================================================
	// Company        : LogTech, s.r.o.
	// Created by     : Mahmoud Elnady
	// Block          : OPC_SendReciveAck
	// Project        : Lekarna, Chrudim -PLC001 -MCC001
	// Project number : 23-157
	// ==========================================================================================================================================
	
	//======================================================
	// Region: Communication Handling and Logging
	// Description: Manages the communication routine and logs
	//              events for message sending, acknowledgment
	//              reception, and acknowledgment timeout.
	//======================================================
	   
	//------------------------------------------------------
	// Call communication routine
	//------------------------------------------------------
	REGION Communication Routine
	    #Comm(SourceSeq := #staSource.SourceSeq,
	          AckSeq := #staAck.AckSeq,
	             Timeout := T#20s);
	END_REGION
	
	#Source.SourceSeq := #staSource.SourceSeq;
	#staAck.AckSeq := #Ack.AckSeq;
	
	
	//------------------------------------------------------
	// Log event when a new message is sent
	//------------------------------------------------------
	REGION Log event - new message
	    IF #Comm.Log.Send THEN
	        #Comm.Log.Send := FALSE;
	        
	        // (LOG)3001=$ Node $, new message sent, seq: $, $ $ $ $ $ $ $ $, $ $ $ $ $ $ $ $ $ $ $ $ $ $ $ $
	        DB_LogMsg.LogMsg_1.Para_BYTE_02.Data := #Source.SourceSeq;
	        
	        // Call logging function
	        #Retval := FC_LogMsg(EventID := 3007,
	                               EventLevel := 2,
	                               EventGroup := 33,
	                               LogMsg := DB_LogMsg.LogMsg_1);
	    END_IF;
	END_REGION
	
	   
	//------------------------------------------------------
	// Log event when new acknowledgment is received
	//------------------------------------------------------
	REGION  Log event-New acknowledgment
	       IF #Comm.Log.New_Ack_received THEN
	           #Comm.Log.New_Ack_received := FALSE;
	           
	           // (LOG)3008=$ Node $, acknowledge received, seq: $, WMSID: $
	           DB_LogMsg.LogMsg_2.Para_BYTE_02.Data := #Ack.AckSeq;
	           
	           // Call logging function
	           #Retval := FC_LogMsg(EventID := 3008,
	                                  EventLevel := 2,
	                                  EventGroup := 33,
	                                  LogMsg := DB_LogMsg.LogMsg_2);
	       END_IF;
	END_REGION
	
	   
	//------------------------------------------------------
	// Log event when acknowledgment timeout occurs
	//------------------------------------------------------
	REGION Log event- acknowledgment timeout
	       IF #Comm.Log.Ack_timeout THEN
	           #Comm.Log.Ack_timeout := FALSE;
	           
	           // (LOG)3009=$ Node $, seq: $, acknowledge timeout!
	           DB_LogMsg.LogMsg_3.Para_BYTE_02.Data := #Comm.SendSeq;
	           
	           // Call logging function
	           #Retval := FC_LogMsg(EventID := 3009,
	                                  EventLevel := 3,
	                                  EventGroup := 33,
	                                  LogMsg := DB_LogMsg.LogMsg_3);
	       END_IF;
	END_REGION
	    
	
	   
	   
	
END_FUNCTION_BLOCK
END_NAMESPACE

NAMESPACE ProductionLine
FUNCTION_BLOCK FB_Segments
{ S7_Optimized_Access := 'TRUE' ; Published := 'FALSE' }
VERSION : 0.1
   VAR 
      ConveyorID : Int;
      "Counter" : Int;
      FlowRackLoop1 : Array[_."B1.1.1".._."B1.23.1"] of Bool;
      FlowRackLoop2 : Array[_."B1.6.1".._."B1.18.1"] of Bool;
      Fragileloop1 : Array[_."D1.1.1".._."E1.6.1"] of Bool;
      Fragileloop2 : Array[_."D1.9.1".._."D1.10.1"] of Bool;
      cmp : Struct
         FlowRackLoop1 : Array[_."B1.1.1".._."B1.23.1"] of Bool;
         FlowRackLoop2 : Array[_."B1.6.1".._."B1.18.1"] of Bool;
         Fragileloop1 : Array[_."D1.1.1".._."E1.6.1"] of Bool;
         Fragileloop2 : Array[_."D1.9.1".._."D1.10.1"] of Bool;
      END_STRUCT;
      FlowRackLoopReadyToRun : Bool;
      FlowRackWorkPlaceLeftReadyToRun : Bool;
      FlowRackWorkPlaceRightReadyToRun : Bool;
      FragileloopReadyToRun : Bool;
   END_VAR


BEGIN
	// ==========================================================================================================================================
	// Company        : LogTech, s.r.o.
	// Created by     : Mahmoud Elnady
	// Block          : FB_Segments
	// Project        : Lekarna, Chrudim -PLC001 -MCC001
	// Project number : 23-157
	// ==========================================================================================================================================
	
	// ===============================
	// REGION: Flow rack loop
	// Purpose: Check the ReadyToRun status of conveyors and transfer units 
	//          for a flow rack section, then compare with a stored snapshot.
	// ===============================
	REGION Flow rack loop
	    
	    // ---------------------------------
	    // REGION: Conveyor Status Loop
	    // Purpose: Iterate over conveyor IDs from B1.1.1 to B1.28.1 
	    //          and store their ReadyToRun status in FlowRackLoop1 array.
	    // ---------------------------------
	   REGION Conveyor Status
	        FOR #Counter := _."B1.1.1" TO _."B1.23.1" DO
	            // Store ReadyToRun status of the current conveyor into FlowRackLoop1
	            #FlowRackLoop1[#Counter] := 
	            _.Global.DB_Global.Status.Line.ProductionLine.ReadyToRun[#Counter];
	        END_FOR;
	    END_REGION
	   
	    // ---------------------------------
	    // REGION: Transfer Unit Status Loop
	    // Purpose: Iterate over transfer unit IDs from B1.6.1 to B1.21.1 
	    //          and store their ReadyToRun status in FlowRackLoop2 array.
	    // ---------------------------------
	    REGION TransferUnit Status
	        FOR #Counter := _."B1.6.1" TO _."B1.18.1" DO
	            // Store ReadyToRun status of the current transfer unit into FlowRackLoop2
	            #FlowRackLoop2[#Counter] :=
	            _.Global.DB_Global.Status.Line.ProductionLine.ReadyToRun[#Counter];
	        END_FOR;
	    END_REGION
	    
	    // ---------------------------------
	    // REGION: Status Comparison
	    // Purpose: Check if both conveyor and transfer unit statuses 
	    //          match the previous recorded values (#cmp arrays).
	    // ---------------------------------
	    REGION Comparison
	        #FlowRackLoopReadyToRun := NOT 
	        ((#cmp.FlowRackLoop1 = #FlowRackLoop1) AND
	        (#cmp.FlowRackLoop2 = #FlowRackLoop2));
	    END_REGION
	    
	END_REGION
	
	
	// ===============================
	// REGION: Flow rack work place left
	// Purpose: ReadyToRun check for two specific conveyors on the left side.
	// ===============================
	REGION Flow rack work place left
	    #FlowRackWorkPlaceLeftReadyToRun :=
	    _.Global.DB_Global.Status.Line.ProductionLine.ReadyToRun[_."C1.4.1"] AND
	    _.Global.DB_Global.Status.Line.ProductionLine.ReadyToRun[_."C1.4.2"];
	END_REGION
	
	
	// ===============================
	// REGION: Flow rack work place right
	// Purpose: ReadyToRun check for two specific conveyors on the right side.
	// ===============================
	REGION Flow rack work place right
	    #FlowRackWorkPlaceRightReadyToRun :=
	    _.Global.DB_Global.Status.Line.ProductionLine.ReadyToRun[_."C1.2.1"] AND
	    _.Global.DB_Global.Status.Line.ProductionLine.ReadyToRun[_."C1.2.2"];
	END_REGION
	
	
	// ===============================
	// REGION: Fragile loop
	// Purpose: Same logic as Flow rack loop, but for the "fragile" product path.
	// ===============================
	REGION Fragile loop
	    
	    // ---------------------------------
	    // REGION: Conveyor Status Loop (Fragile)
	    // Purpose: Store ReadyToRun status for conveyors D1.1.1 to E1.6.1
	    // ---------------------------------
	    REGION Conveyor Status
	        FOR #Counter := _."D1.1.1" TO _."E1.6.1" DO
	            #Fragileloop1[#Counter] :=
	            _.Global.DB_Global.Status.Line.ProductionLine.ReadyToRun[#Counter];
	        END_FOR;
	    END_REGION
	    
	    // ---------------------------------
	    // REGION: Transfer Unit Status Loop (Fragile)
	    // Purpose: Store ReadyToRun status for transfer units D1.8.1 to D1.9.1
	    // ---------------------------------
	    REGION TransferUnit Status
	        FOR #Counter := _."D1.9.1" TO _."D1.10.1" DO
	            #Fragileloop2[#Counter] :=
	            _.Global.DB_Global.Status.Line.ProductionLine.ReadyToRun[#Counter];
	        END_FOR;
	    END_REGION
	    
	    // ---------------------------------
	    // REGION: Status Comparison (Fragile)
	    // Purpose: Check if current fragile loop status matches previous snapshot.
	    // ---------------------------------
	    REGION Comparison
	        #FragileloopReadyToRun := NOT
	        ((#cmp.Fragileloop1 = #Fragileloop1) AND
	        (#cmp.Fragileloop2 = #Fragileloop2));
	    END_REGION
	    
	END_REGION
	
END_FUNCTION_BLOCK
END_NAMESPACE

NAMESPACE ProductionLine
FUNCTION_BLOCK FB_Technology
{ S7_Optimized_Access := 'TRUE' ; Published := 'FALSE' }
VERSION : 0.1
   VAR 
      IP11 : String := 'IP11';
      IP12 : String := 'IP12';
      IP21 : String := 'IP21';
      IP22 : String := 'IP22';
      IP23 : String := 'IP23';
      IP31 : String := 'IP31';
      IP32 : String := 'IP32';
      IP41 : String := 'IP41';
      IP42 : String := 'IP42';
      ComDownStream : Struct
         DP1 : Bool;
         DP2 : Bool;
         DP3 : Bool;
         DP4 : Bool;
      END_STRUCT;
      ComTimmerDP1 {InstructionName := 'TON_TIME'; LibVersion := '1.0'} : TON_TIME;
      ComTimmerDP2 {InstructionName := 'TON_TIME'; LibVersion := '1.0'} : TON_TIME;
      ComTimmerDP3 {InstructionName := 'TON_TIME'; LibVersion := '1.0'} : TON_TIME;
      ComTimmerDP4 {InstructionName := 'TON_TIME'; LibVersion := '1.0'} : TON_TIME;
   END_VAR


BEGIN
	// ==========================================================================================================================================
	// Company        : LogTech, s.r.o.
	// Created by     : Mahmoud Elnady
	// Block          : FB_OPC_Communication
	// Project        : Lekarna, Chrudim -PLC001 -MCC001
	// Project number : 23-157
	// ==========================================================================================================================================
	
	REGION Destination request TO WMS
	    // Send destination request to WMS
	    REGION DP1
	        IF IDB_BarcodeReader.DP1."Dataman-Results Available" OR
	            IDB_ProductionLine."A1.5.1".CONVEYOR_SENSOR.PosEdge.Q
	        THEN
	            OPC_Data.DP1.DestRequest.Source.Barcode := IDB_BarcodeReader.DP1.ResultStr;
	            IDB_OPC_Communication.Communication_DP1.Communication.Send := TRUE;
	            #ComDownStream.DP1 := TRUE;
	        ELSIF (IDB_OPC_Communication.Communication_DP1.Communication.SourceSeq =
	            IDB_OPC_Communication.Communication_DP1.Communication.AckSeq)
	            OR #ComTimmerDP1.Q
	        THEN
	            IDB_OPC_Communication.Communication_DP1.Communication.Send := FALSE;
	        END_IF;
	         
	    END_REGION
	    
	    REGION DP2
	        IF IDB_BarcodeReader.DP2."Dataman-Results Available" OR
	            IDB_ProductionLine."B1.9.1".CONVEYOR_SENSOR.PosEdge.Q
	        THEN
	            OPC_Data.DP2.DestRequest.Source.Barcode := IDB_BarcodeReader.DP2.ResultStr;
	            IDB_OPC_Communication.Communication_DP2.Communication.Send := TRUE;
	            #ComDownStream.DP2 := TRUE;
	        ELSIF (IDB_OPC_Communication.Communication_DP2.Communication.SourceSeq =
	            IDB_OPC_Communication.Communication_DP2.Communication.AckSeq)
	            OR #ComTimmerDP2.Q
	        THEN
	            IDB_OPC_Communication.Communication_DP2.Communication.Send := FALSE;
	        END_IF;
	    END_REGION
	    
	    REGION DP3
	        IF IDB_BarcodeReader.DP3."Dataman-Results Available" OR
	            IDB_ProductionLine."B1.17.1".CONVEYOR_SENSOR.PosEdge.Q
	        THEN
	            OPC_Data.DP3.DestRequest.Source.Barcode := IDB_BarcodeReader.DP3.ResultStr;
	            IDB_OPC_Communication.Communication_DP3.Communication.Send := TRUE;
	            #ComDownStream.DP3 := TRUE;
	        ELSIF (IDB_OPC_Communication.Communication_DP3.Communication.SourceSeq =
	            IDB_OPC_Communication.Communication_DP3.Communication.AckSeq)
	            OR #ComTimmerDP3.Q
	        THEN
	            IDB_OPC_Communication.Communication_DP3.Communication.Send := FALSE;
	        END_IF;
	    END_REGION
	    
	    REGION DP4
	        IF IDB_BarcodeReader.DP4."Dataman-Results Available" OR
	            IDB_ProductionLine."A1.7.4".CONVEYOR_SENSOR.PosEdge.Q
	        THEN
	            OPC_Data.DP4.DestRequest.Source.Barcode := IDB_BarcodeReader.DP4.ResultStr;
	            IDB_OPC_Communication.Communication_DP4.Communication.Send := TRUE;
	            #ComDownStream.DP4 := TRUE;
	        ELSIF (IDB_OPC_Communication.Communication_DP4.Communication.SourceSeq =
	            IDB_OPC_Communication.Communication_DP4.Communication.AckSeq)
	            OR #ComTimmerDP4.Q
	        THEN
	            IDB_OPC_Communication.Communication_DP4.Communication.Send := FALSE;
	        END_IF;
	        
	    END_REGION
	    
	END_REGION
	
	REGION Wait FOR data from WMS
	    // Wait for data from WMS
	    REGION Mabs A1.6.1 & A1.6.2 Dir
	        IF IDB_OPC_Communication.Communication_DP1.Communication.New_Ack_received THEN
	            //IDB_OPC_Communication.Communication_DP1.Communication.New_Ack_received := FALSE;
	            #ComDownStream.DP1 := FALSE;
	            IF OPC_Data.DP1.DestRequest.Ack.Destination = #IP11 THEN
	                DB_ToteTracking.Conveyor[_."A1.5.1"].ToteDir.Straight := TRUE;
	                DB_ToteTracking.Conveyor[_."A1.5.1"].ToteDir.toRight := FALSE;
	                DB_ToteTracking.Conveyor[_."A1.2.1"].ToteDir.toLeft := FALSE;
	            ELSIF
	                OPC_Data.DP1.DestRequest.Ack.Destination = #IP12 THEN
	                DB_ToteTracking.Conveyor[_."A1.5.1"].ToteDir.toRight := TRUE;
	                DB_ToteTracking.Conveyor[_."A1.5.1"].ToteDir.Straight := FALSE;
	                DB_ToteTracking.Conveyor[_."A1.5.1"].ToteDir.toLeft := FALSE;
	            ELSE
	                DB_ToteTracking.Conveyor[_."A1.5.1"].ToteDir.Straight := FALSE;
	                DB_ToteTracking.Conveyor[_."A1.5.1"].ToteDir.toRight := FALSE;
	                DB_ToteTracking.Conveyor[_."A1.5.1"].ToteDir.toLeft := FALSE;
	            END_IF;
	        END_IF;
	    END_REGION
	    
	    REGION Transfer Unit B1.10.1 Dir
	        IF IDB_OPC_Communication.Communication_DP2.Communication.New_Ack_received THEN
	            //IDB_OPC_Communication.Communication_DP2.Communication.New_Ack_received := FALSE;
	            #ComDownStream.DP2 := FALSE;
	            IF  OPC_Data.DP2.DestRequest.Ack.Destination = #IP21 THEN
	                DB_ToteTracking.Conveyor[_."B1.9.1"].ToteDir.Straight := TRUE;
	                DB_ToteTracking.Conveyor[_."B1.9.1"].ToteDir.toRight := FALSE;
	                DB_ToteTracking.Conveyor[_."B1.9.1"].ToteDir.toLeft := FALSE;
	            ELSIF
	                (OPC_Data.DP2.DestRequest.Ack.Destination = #IP22 OR
	                OPC_Data.DP2.DestRequest.Ack.Destination = #IP23) THEN
	                DB_ToteTracking.Conveyor[_."B1.9.1"].ToteDir.toRight := TRUE;
	                DB_ToteTracking.Conveyor[_."B1.9.1"].ToteDir.Straight := FALSE;
	                DB_ToteTracking.Conveyor[_."B1.9.1"].ToteDir.toLeft := FALSE;
	                //Transfer Unit C1.1.3 Dir
	                IF OPC_Data.DP2.DestRequest.Ack.Destination = #IP22 THEN
	                    DB_ToteTracking.Transfer[_."B1.9.1"].Straight := FALSE;
	                    DB_ToteTracking.Transfer[_."B1.9.1"].toRight := TRUE;
	                    DB_ToteTracking.Transfer[_."B1.9.1"].toLeft := FALSE;
	                ELSIF  OPC_Data.DP2.DestRequest.Ack.Destination = #IP23 THEN
	                    DB_ToteTracking.Transfer[_."B1.9.1"].toRight := FALSE;
	                    DB_ToteTracking.Transfer[_."B1.9.1"].Straight := FALSE;
	                    DB_ToteTracking.Transfer[_."B1.9.1"].toLeft := TRUE;
	                ELSE
	                    DB_ToteTracking.Transfer[_."B1.9.1"].Straight := FALSE;
	                    DB_ToteTracking.Transfer[_."B1.9.1"].toRight := FALSE;
	                    DB_ToteTracking.Transfer[_."B1.9.1"].toLeft := FALSE;
	                END_IF;
	                
	            ELSE
	                DB_ToteTracking.Conveyor[_."B1.9.1"].ToteDir.Straight := FALSE;
	                DB_ToteTracking.Conveyor[_."B1.9.1"].ToteDir.toRight := FALSE;
	                DB_ToteTracking.Conveyor[_."B1.9.1"].ToteDir.toLeft := FALSE;
	            END_IF;
	        END_IF;
	    END_REGION
	    
	    
	    REGION Transfer Unit B1.21.1 Dir
	        IF IDB_OPC_Communication.Communication_DP3.Communication.New_Ack_received THEN
	            //IDB_OPC_Communication.Communication_DP3.Communication.New_Ack_received := FALSE;
	            #ComDownStream.DP3 := FALSE;
	            IF  OPC_Data.DP3.DestRequest.Ack.Destination = #IP31 THEN
	                DB_ToteTracking.Conveyor[_."B1.17.1"].ToteDir.Straight := TRUE;
	                DB_ToteTracking.Conveyor[_."B1.17.1"].ToteDir.toRight := FALSE;
	                DB_ToteTracking.Conveyor[_."B1.17.1"].ToteDir.toLeft := FALSE;
	                
	            ELSIF OPC_Data.DP3.DestRequest.Ack.Destination = #IP32 THEN
	                DB_ToteTracking.Conveyor[_."B1.17.1"].ToteDir.toRight := FALSE;
	                DB_ToteTracking.Conveyor[_."B1.17.1"].ToteDir.Straight := FALSE;
	                DB_ToteTracking.Conveyor[_."B1.17.1"].ToteDir.toLeft := TRUE;
	                
	            ELSE
	                DB_ToteTracking.Conveyor[_."B1.17.1"].ToteDir.Straight := FALSE;
	                DB_ToteTracking.Conveyor[_."B1.17.1"].ToteDir.toRight := FALSE;
	                DB_ToteTracking.Conveyor[_."B1.17.1"].ToteDir.toLeft := FALSE;
	            END_IF;
	        END_IF;
	    END_REGION
	    
	    REGION Mabs A1.8.1 & A1.8.2 Dir
	        IF IDB_OPC_Communication.Communication_DP4.Communication.New_Ack_received THEN
	            //IDB_OPC_Communication.Communication_DP4.Communication.New_Ack_received := FALSE;
	            #ComDownStream.DP4 := FALSE;
	            IF  OPC_Data.DP4.DestRequest.Ack.Destination = #IP41 THEN
	                DB_ToteTracking.Conveyor[_."A1.7.4"].ToteDir.Straight := TRUE;
	                DB_ToteTracking.Conveyor[_."A1.7.4"].ToteDir.toRight := FALSE;
	                DB_ToteTracking.Conveyor[_."A1.7.4"].ToteDir.toLeft := FALSE;
	            ELSIF
	                OPC_Data.DP4.DestRequest.Ack.Destination = #IP42 THEN
	                DB_ToteTracking.Conveyor[_."A1.7.4"].ToteDir.toRight := TRUE;
	                DB_ToteTracking.Conveyor[_."A1.7.4"].ToteDir.Straight := FALSE;
	                DB_ToteTracking.Conveyor[_."A1.7.4"].ToteDir.toLeft := FALSE;
	            ELSE
	                DB_ToteTracking.Conveyor[_."A1.7.4"].ToteDir.Straight := FALSE;
	                DB_ToteTracking.Conveyor[_."A1.7.4"].ToteDir.toRight := FALSE;
	                DB_ToteTracking.Conveyor[_."A1.7.4"].ToteDir.toLeft := FALSE;
	            END_IF;
	        END_IF;
	    END_REGION
	    
	    REGION Wait WMS Response
	        #ComTimmerDP1(IN := #ComDownStream.DP1,
	                      PT := t#45s);
	        
	        IF #ComTimmerDP1.Q THEN
	            #ComDownStream.DP1 := FALSE;
	        END_IF;
	        
	        #ComTimmerDP2(IN := #ComDownStream.DP2,
	                      PT := t#45s);
	        
	        IF #ComTimmerDP2.Q THEN
	            #ComDownStream.DP2 := FALSE;
	        END_IF;
	        
	        #ComTimmerDP3(IN := #ComDownStream.DP3,
	                      PT := t#45s);
	        
	        IF #ComTimmerDP3.Q THEN
	            #ComDownStream.DP3 := FALSE;
	        END_IF;
	        
	        #ComTimmerDP4(IN := #ComDownStream.DP4,
	                      PT := t#45s);
	        
	        IF #ComTimmerDP4.Q THEN
	            #ComDownStream.DP4 := FALSE;
	        END_IF;
	        
	    END_REGION
	
	END_REGION
	
	
	REGION Destination info TO WMS
	    // Send destination info to WMS
	    REGION IP1
	        IF IDB_ProductionLine."A1.7.2".CONVEYOR_SENSOR.PosEdge.Q AND
	            NOT IDB_OPC_Communication.Communication_IP1.Communication.Send THEN
	            OPC_Data.IP11.DestInfo.Source.Barcode := DB_ToteTracking.Conveyor[_."A1.7.1"].Barcode;
	            OPC_Data.IP11.DestInfo.Source.InformationPoint := #IP11;
	            IDB_OPC_Communication.Communication_IP1.Communication.Send := TRUE;
	        END_IF;
	        
	    END_REGION
	    REGION IP2
	        IF IDB_ProductionLine."B1.2.1".CONVEYOR_SENSOR.PosEdge.Q AND
	            NOT IDB_OPC_Communication.Communication_IP2.Communication.Send THEN
	            OPC_Data.IP12.DestInfo.Source.Barcode := DB_ToteTracking.Conveyor[_."B1.1.1"].Barcode;
	            OPC_Data.IP12.DestInfo.Source.InformationPoint := #IP12;
	            IDB_OPC_Communication.Communication_IP2.Communication.Send := TRUE;
	        END_IF;
	        
	    END_REGION
	    
	    REGION IP3
	        IF IDB_ProductionLine."B1.11.2".CONVEYOR_SENSOR.PosEdge.Q AND
	            NOT IDB_OPC_Communication.Communication_IP3.Communication.Send THEN
	            OPC_Data.IP21.DestInfo.Source.Barcode := DB_ToteTracking.Conveyor[_."B1.11.1"].Barcode;
	            OPC_Data.IP21.DestInfo.Source.InformationPoint := #IP21;
	            IDB_OPC_Communication.Communication_IP3.Communication.Send := TRUE;
	        END_IF;
	    END_REGION
	    
	    REGION IP4
	        IF IDB_ProductionLine."C1.2.1".CONVEYOR_SENSOR.PosEdge.Q AND
	            NOT IDB_OPC_Communication.Communication_IP4.Communication.Send THEN
	            OPC_Data.IP22.DestInfo.Source.Barcode := DB_ToteTracking.Conveyor[_."C1.2.2"].Barcode;
	            OPC_Data.IP22.DestInfo.Source.InformationPoint := #IP22;
	            IDB_OPC_Communication.Communication_IP4.Communication.Send := TRUE;
	        END_IF;
	        
	    END_REGION
	    
	    REGION IP5
	        IF IDB_ProductionLine."C1.4.2".CONVEYOR_SENSOR.PosEdge.Q AND
	            NOT IDB_OPC_Communication.Communication_IP5.Communication.Send THEN
	            OPC_Data.IP23.DestInfo.Source.Barcode := DB_ToteTracking.Conveyor[_."C1.4.1"].Barcode;
	            OPC_Data.IP23.DestInfo.Source.InformationPoint := #IP23;
	            IDB_OPC_Communication.Communication_IP5.Communication.Send := TRUE;
	        END_IF;
	        
	    END_REGION
	    
	    REGION IP6
	        IF IDB_ProductionLine."B1.20.1".CONVEYOR_SENSOR.PosEdge.Q AND
	            NOT IDB_OPC_Communication.Communication_IP6.Communication.Send THEN
	            OPC_Data.IP31.DestInfo.Source.Barcode := DB_ToteTracking.Conveyor[_."B1.19.1"].Barcode;
	            OPC_Data.IP31.DestInfo.Source.InformationPoint := #IP31;
	            IDB_OPC_Communication.Communication_IP6.Communication.Send := TRUE;
	        END_IF;
	    END_REGION
	    
	    REGION IP7
	        IF (IDB_S300_FullControl."Left/RightSensor" OR
	            IDB_Flow_Test.R_TRIG_Instance.Q) AND //only for simulation purpose 
	            NOT IDB_OPC_Communication.Communication_IP7.Communication.Send THEN
	            OPC_Data.IP32.DestInfo.Source.Barcode := DB_ToteTracking.Conveyor[_."B1.6.1"].Barcode;
	            OPC_Data.IP32.DestInfo.Source.InformationPoint := #IP32;
	            IDB_OPC_Communication.Communication_IP7.Communication.Send := TRUE;
	        END_IF;
	        
	    END_REGION
	    
	    REGION IP8
	        IF IDB_ProductionLine."A1.10.2".CONVEYOR_SENSOR.PosEdge.Q AND
	            NOT IDB_OPC_Communication.Communication_IP8.Communication.Send THEN
	            OPC_Data.IP41.DestInfo.Source.Barcode := DB_ToteTracking.Conveyor[_."A1.10.1"].Barcode;
	            OPC_Data.IP41.DestInfo.Source.InformationPoint := #IP41;
	            IDB_OPC_Communication.Communication_IP8.Communication.Send := TRUE;
	        END_IF;
	    END_REGION
	    
	    REGION IP9
	        IF IDB_ProductionLine."D1.2.1".CONVEYOR_SENSOR.PosEdge.Q AND
	            NOT IDB_OPC_Communication.Communication_IP9.Communication.Send THEN
	            OPC_Data.IP42.DestInfo.Source.Barcode := DB_ToteTracking.Conveyor[_."D1.1.1"].Barcode;
	            OPC_Data.IP42.DestInfo.Source.InformationPoint := #IP42;
	            IDB_OPC_Communication.Communication_IP9.Communication.Send := TRUE;
	        END_IF;
	    END_REGION
	    
	    
	END_REGION
	
	
	REGION Wait FOR data from WMS
	    // Wait for data from WMS
	    REGION IP1 Ack
	        IF IDB_OPC_Communication.Communication_IP1.Communication.New_Ack_received THEN
	            IDB_OPC_Communication.Communication_IP1.Communication.Send := FALSE;
	            IDB_OPC_Communication.Communication_IP1.Communication.New_Ack_received := FALSE;
	        END_IF;
	    END_REGION
	    
	    REGION IP2 Ack
	        IF IDB_OPC_Communication.Communication_IP2.Communication.New_Ack_received THEN
	            IDB_OPC_Communication.Communication_IP2.Communication.Send := FALSE;
	            IDB_OPC_Communication.Communication_IP2.Communication.New_Ack_received := FALSE;
	        END_IF;
	    END_REGION
	    
	    REGION IP3 Ack
	        IF IDB_OPC_Communication.Communication_IP3.Communication.New_Ack_received THEN
	            IDB_OPC_Communication.Communication_IP3.Communication.Send := FALSE;
	            IDB_OPC_Communication.Communication_IP3.Communication.New_Ack_received := FALSE;
	        END_IF;
	    END_REGION
	    
	    REGION IP4 Ack
	        IF IDB_OPC_Communication.Communication_IP4.Communication.New_Ack_received THEN
	            IDB_OPC_Communication.Communication_IP4.Communication.Send := FALSE;
	            IDB_OPC_Communication.Communication_IP4.Communication.New_Ack_received := FALSE;
	        END_IF;
	    END_REGION
	    
	    REGION IP5 Ack
	        IF IDB_OPC_Communication.Communication_IP5.Communication.New_Ack_received THEN
	            IDB_OPC_Communication.Communication_IP5.Communication.Send := FALSE;
	            IDB_OPC_Communication.Communication_IP5.Communication.New_Ack_received := FALSE;
	        END_IF;
	    END_REGION
	    
	    REGION IP6 Ack
	        IF IDB_OPC_Communication.Communication_IP6.Communication.New_Ack_received THEN
	            IDB_OPC_Communication.Communication_IP6.Communication.Send := FALSE;
	            IDB_OPC_Communication.Communication_IP6.Communication.New_Ack_received := FALSE;
	        END_IF;
	    END_REGION
	    
	    REGION IP7 Ack
	        IF IDB_OPC_Communication.Communication_IP7.Communication.New_Ack_received THEN
	            IDB_OPC_Communication.Communication_IP7.Communication.Send := FALSE;
	            IDB_OPC_Communication.Communication_IP7.Communication.New_Ack_received := FALSE;
	        END_IF;
	    END_REGION
	    
	    REGION IP8 Ack
	        IF IDB_OPC_Communication.Communication_IP8.Communication.New_Ack_received THEN
	            IDB_OPC_Communication.Communication_IP8.Communication.Send := FALSE;
	            IDB_OPC_Communication.Communication_IP8.Communication.New_Ack_received := FALSE;
	        END_IF;
	    END_REGION
	    
	    REGION IP9 Ack
	        IF IDB_OPC_Communication.Communication_IP9.Communication.New_Ack_received THEN
	            IDB_OPC_Communication.Communication_IP9.Communication.Send := FALSE;
	            IDB_OPC_Communication.Communication_IP9.Communication.New_Ack_received := FALSE;
	        END_IF;
	    END_REGION
	    
	END_REGION
	
	
	
	
	
	
	
	
	
	   
	        
	         
END_FUNCTION_BLOCK
END_NAMESPACE

NAMESPACE ProductionLine
FUNCTION FC_LogMsg : Int
{ S7_Optimized_Access := 'TRUE' ; Published := 'FALSE' }
VERSION : 0.1
   VAR_INPUT 
      EventID : Int;
      EventLevel : Byte;
      EventGroup : Byte;
      LogMsg : Variant;
   END_VAR

   VAR_TEMP 
      LtLogMsg : Log_LogMsg_Header;
      LabyAuxBuffer : Array[0..1023] of Byte;
      LdiMsgPosition : DInt;
      LdiMsgStartPosition : DInt;
      LiReturn : Int;
   END_VAR

   VAR CONSTANT 
      coSTX : Byte := 16#2;
      coSOH : Byte := 16#1;
      coMsgType_Log : Byte := 16#5;
      LOGMSG_BUFFER_SIZE : Int := 8191;
   END_VAR


BEGIN
	// ==========================================================================================================================================
	// Company        : LogTech, s.r.o.
	// Created by     : Mahmoud Elnady
	// Block          : OPC_SendReciveAck
	// Project        : Lekarna, Chrudim -PLC001 -MCC001
	// Project number : 23-157
	// ==========================================================================================================================================
	
	
	#LtLogMsg.STX := #coSTX;                              // initialisation of fixed header fields
	#LtLogMsg.SOH := #coSOH;
	#LtLogMsg.MsgType := #coMsgType_Log;
	
	#LtLogMsg.EventLevel := #EventLevel;                 // write input parameters into message header
	#LtLogMsg.EventGroup := #EventGroup;
	#LtLogMsg.EventID := #EventID;
	
	#LtLogMsg.MsgLength := 0;                               // initialisation of message length in header
	#LdiMsgPosition := 0;                                   // initialisation of write position in auxiliary buffer
	
	// !!! how to get timestamp with less cycle time consumption ???
	#LiReturn := RD_LOC_T(#LtLogMsg.Timestamp);            // write system date and time into message header
	
	// write message header into auxiliary buffer (message length in header still invalid!)
	#FC_LogMsg := Serialize(SRC_VARIABLE := #LtLogMsg, DEST_ARRAY => #LabyAuxBuffer, POS := #LdiMsgPosition);
	IF #FC_LogMsg <> 0 THEN
	    RETURN;                 // instruction faulted - error status returned in iRetVal
	END_IF;
	
	// write message data into auxiliary buffer
	#FC_LogMsg := Serialize(SRC_VARIABLE := #LogMsg, DEST_ARRAY => #LabyAuxBuffer, POS := #LdiMsgPosition);
	IF #FC_LogMsg <> 0 THEN
	    RETURN;                 // instruction faulted - error status returned in iRetVal
	END_IF;
	
	// check if the message data fits in the buffer
	IF DB_LogMsg.Write_Position + DINT_TO_INT(#LdiMsgPosition) > #LOGMSG_BUFFER_SIZE THEN
	    RETURN;
	END_IF;
	
	#LtLogMsg.MsgLength := DINT_TO_INT(#LdiMsgPosition);    // write message length into message header
	
	#LabyAuxBuffer[2] := #LtLogMsg.MsgLength.%B0;            // and write it bytewise into appropriate position in auxiliary buffer
	#LabyAuxBuffer[3] := #LtLogMsg.MsgLength.%B1;
	
	// ^^^ REPLACED with previous lines ^^^
	// overwrite the message header in buffer with valid message length
	// #LogMsg := Serialize(SRC_VARIABLE := #tHeader, DEST_ARRAY => "LogMsg_DB".abyLogMsg_Buffer, POS := #LdiMsgStartPosition);
	// IF #LogMsg <> 0 THEN
	//     RETURN;                 // instruction faulted - error status returned in iRetVal
	// END_IF;
	
	// ! INTERRUPT DISABLED !
	#LiReturn := DIS_IRT(MODE := 0, OB_NR := 0);
	
	MOVE_BLK(IN := #LabyAuxBuffer[0],
	         COUNT := DINT_TO_ULINT(#LdiMsgPosition),
	         OUT => DB_LogMsg.abyLogMsg_Buffer[DB_LogMsg.Write_Position]);
	
	DB_LogMsg.Write_Position := DB_LogMsg.Write_Position + DINT_TO_INT(#LdiMsgPosition);    // if everything was ok, update the write position in buffer
	
	// ! INTERRUPT ENABLE !
	#LiReturn := EN_IRT(MODE := 0, OB_NR := 0);
	
	// !!! all messages since last send are in "LogMsg_DB".abyLogMsg_Buffer - somewhere must be function to send these data to log server
	// !!! is this safe for interrupt(s) ? and optimal ?
	// !!! what about sequence number ? should we have one ?
	// !!! solution for buffer overflow !
	
END_FUNCTION
END_NAMESPACE

NAMESPACE ProductionLine
FUNCTION_BLOCK FB_ToteTracking
{ S7_Optimized_Access := 'TRUE' ; Published := 'FALSE' }
VERSION : 0.1
   VAR 
      ZoneBpJam_Occ {InstructionName := 'TON_TIME'; LibVersion := '1.0'; S7_SetPoint := 'False'} : TON_TIME;
      ZoneBpJam_NotOcc {InstructionName := 'TON_TIME'; LibVersion := '1.0'} : TON_TIME;
      DivertToManual { S7_SetPoint := 'True'} : Bool;
      HoldDivertToManual : Bool;
      "RT_Exit_1_" {InstructionName := 'R_TRIG'; LibVersion := '1.0'; S7_SetPoint := 'False'} : Array[1..1] of R_TRIG;
      "RT_Exit_2_" {InstructionName := 'R_TRIG'; LibVersion := '1.0'; S7_SetPoint := 'False'} : Array[1..6] of R_TRIG;
      NoReadTote { S7_SetPoint := 'True'} : String := 'BOX-9999-99999';
      NoData : Array[1..6] of Bool;
   END_VAR


BEGIN
	// ==========================================================================================================================================
	// Company        : LogTech, s.r.o.
	// Created by     : Anton Vinoth Soundraraj
	// Block          : FB_CreatePostData
	// Project        : Gurkerl, Vienna -PLC001 -MCC100
	// Project number : 23-158
	// ==========================================================================================================================================
	
	REGION A1.5.1
	    
	    // write barcode data
	    DB_ToteTracking.Conveyor[_."A1.5.1"].Barcode :=
	    IDB_BarcodeReader.DP1.ResultStr;
	    
	END_REGION
	
	
	REGION A1.5.2
	    
	    IF IDB_ProductionLine."A1.5.1".CONVEYOR_SENSOR.SensorEdge.Negative THEN
	        // Barcode
	        DB_ToteTracking.Conveyor[_."A1.5.2"].Barcode :=
	        DB_ToteTracking.Conveyor[_."A1.5.1"].Barcode;
	        // main diverter direction
	        DB_ToteTracking.Conveyor[_."A1.5.2"].ToteDir :=
	        DB_ToteTracking.Conveyor[_."A1.5.1"].ToteDir;
	    END_IF;
	    
	END_REGION
	
	
	REGION A1.5.3
	    
	    IF IDB_ProductionLine."A1.5.2".CONVEYOR_SENSOR.SensorEdge.Negative
	    THEN
	        // Barcode
	        DB_ToteTracking.Conveyor[_."A1.5.3"].Barcode :=
	        DB_ToteTracking.Conveyor[_."A1.5.2"].Barcode;
	        // main diverter direction
	        DB_ToteTracking.Conveyor[_."A1.5.3"].ToteDir :=
	        DB_ToteTracking.Conveyor[_."A1.5.2"].ToteDir;
	    END_IF;
	    
	    
	    REGION Decision: main diverter: before Mabs
	        
	        // to Right
	        IF DB_ToteTracking.Conveyor[_."A1.5.3"].ToteDir.toRight OR
	            (DB_ToteTracking.Conveyor[_."A1.5.3"].Barcode = #NoReadTote) OR // bad read tote
	            _.Global.IDB_HardwareDiag."Cognex -10.106.129.24".CommunicationError // Cognex reader communcation error
	        THEN
	            DB_ToteTracking.Conveyor[_."A1.6.1"].ToteDir.Straight := FALSE;
	            DB_ToteTracking.Conveyor[_."A1.6.1"].ToteDir.toRight := TRUE;
	            DB_ToteTracking.Conveyor[_."A1.6.2"].ToteDir.Straight := FALSE;
	            DB_ToteTracking.Conveyor[_."A1.6.2"].ToteDir.toRight := TRUE;
	        END_IF;
	        // to straight
	        IF DB_ToteTracking.Conveyor[_."A1.5.3"].ToteDir.Straight AND
	            NOT (DB_ToteTracking.Conveyor[_."A1.5.3"].Barcode = #NoReadTote) AND // good read tote
	            NOT _.Global.IDB_HardwareDiag."Cognex -10.106.129.24".CommunicationError // Keyence reader communcation error
	        THEN
	            DB_ToteTracking.Conveyor[_."A1.6.1"].ToteDir.Straight := TRUE;
	            DB_ToteTracking.Conveyor[_."A1.6.1"].ToteDir.toRight := FALSE;
	            DB_ToteTracking.Conveyor[_."A1.6.2"].ToteDir.Straight := TRUE;
	            DB_ToteTracking.Conveyor[_."A1.6.2"].ToteDir.toRight := FALSE;
	        END_IF;
	        
	    END_REGION
	    
	END_REGION
	
	REGION B1.1.1 Right
	    
	    IF  //IDB_ProductionLine."A1.6.1".CROSS_SENSOR_FILTER.SensorEdge.Negative AND
	        IDB_ProductionLine."A1.6.1".CROSS_SENSOR_FILTER.NegEdge.Q AND
	        NOT IDB_ProductionLine."A1.6.1".CurrentPosition.right AND // remove not
	        NOT IDB_ProductionLine."A1.6.2".CurrentPosition.right //AND // remove not
	        //NOT IDB_ProductionLine."B1.1.1".ReadConveyorStatus.Occupied 
	    THEN
	        // Barcode
	        DB_ToteTracking.Conveyor[_."B1.1.1"].Barcode :=
	        DB_ToteTracking.Conveyor[_."A1.5.3"].Barcode;
	    END_IF;
	    
	END_REGION
	
	REGION B1.2.1
	    
	    IF  IDB_ProductionLine."B1.1.1".CONVEYOR_SENSOR.SensorEdge.Negative THEN
	        DB_ToteTracking.Conveyor[_."B1.2.1"] :=DB_ToteTracking.Conveyor[_."B1.1.1"];
	    END_IF;
	    
	END_REGION
	
	REGION B1.3.1
	    
	    IF IDB_ProductionLine."B1.2.1".CONVEYOR_SENSOR.SensorEdge.Negative THEN
	        DB_ToteTracking.Conveyor[_."B1.3.1"] := DB_ToteTracking.Conveyor[_."B1.2.1"];
	    END_IF;
	    
	END_REGION
	
	
	REGION A1.7.1 Straight
	    
	    IF  IDB_ProductionLine."A1.6.1".CROSS_SENSOR_FILTER.SensorEdge.Negative AND
	        NOT IDB_ProductionLine."A1.6.1".CurrentPosition.straight AND  //remove Not
	        NOT IDB_ProductionLine."A1.6.2".CurrentPosition.straight //AND  // remove Not
	        //NOT IDB_ProductionLine."A1.7.1".ReadConveyorStatus.Occupied
	    THEN
	        // Barcode
	        DB_ToteTracking.Conveyor[_."A1.7.1"].Barcode :=
	        DB_ToteTracking.Conveyor[_."A1.5.3"].Barcode;
	    END_IF;
	    
	END_REGION
	
	REGION A1.7.2
	    
	    IF IDB_ProductionLine."A1.7.1".CONVEYOR_SENSOR.SensorEdge.Negative THEN
	        DB_ToteTracking.Conveyor[_."A1.7.2"] := DB_ToteTracking.Conveyor[_."A1.7.1"];
	    END_IF;
	    
	END_REGION
	
	REGION A1.7.3
	    
	    IF IDB_ProductionLine."A1.7.2".CONVEYOR_SENSOR.SensorEdge.Negative THEN
	        DB_ToteTracking.Conveyor[_."A1.7.3"] := DB_ToteTracking.Conveyor[_."A1.7.2"];
	    END_IF;
	    
	END_REGION
	
	/////////////////////////////////////////////////////////
	//DP2
	////////////////////////////////////////////////////////
	
	REGION B1.9.1
	    
	    // write barcode data
	    DB_ToteTracking.Conveyor[_."B1.9.1"].Barcode :=
	    IDB_BarcodeReader.DP2.ResultStr;
	    
	END_REGION
	
	REGION B1.9.2
	    
	    IF IDB_ProductionLine."B1.9.1".CONVEYOR_SENSOR.SensorEdge.Negative
	    THEN
	        // Barcode
	        DB_ToteTracking.Conveyor[_."B1.9.2"].Barcode :=
	        DB_ToteTracking.Conveyor[_."B1.9.1"].Barcode;
	        // main diverter direction
	        DB_ToteTracking.Conveyor[_."B1.9.2"].ToteDir :=
	        DB_ToteTracking.Conveyor[_."B1.9.1"].ToteDir;
	        //
	        DB_ToteTracking.Transfer[_."B1.9.2"] :=
	        DB_ToteTracking.Transfer[_."B1.9.1"];
	    END_IF;
	    
	    
	    REGION Decision: second diverter: before Transfer Unit 
	        
	        // to Right for Transfer Unit B1.10.1
	        IF DB_ToteTracking.Conveyor[_."B1.9.2"].ToteDir.toRight OR
	           (DB_ToteTracking.Conveyor[_."B1.9.2"].Barcode = #NoReadTote) OR // Good read tote
	           _.Global.IDB_HardwareDiag."Cognex -10.106.129.24".CommunicationError // Cognex reader communcation error
	        THEN
	            DB_ToteTracking.Conveyor[_."B1.10.1"].ToteDir.Straight := FALSE;
	            DB_ToteTracking.Conveyor[_."B1.10.1"].ToteDir.toRight := TRUE;
	        END_IF;
	        // to straight for Transfer Unit B1.10.1 
	        IF DB_ToteTracking.Conveyor[_."B1.9.2"].ToteDir.Straight AND
	           NOT (DB_ToteTracking.Conveyor[_."B1.9.2"].Barcode = #NoReadTote) AND // Bad read tote
	           NOT _.Global.IDB_HardwareDiag."Cognex -10.106.129.24".CommunicationError // Cognex reader communcation error
	        THEN
	            DB_ToteTracking.Conveyor[_."B1.10.1"].ToteDir.Straight := TRUE;
	            DB_ToteTracking.Conveyor[_."B1.10.1"].ToteDir.toRight := FALSE;
	        END_IF;
	        
	        // to Right for Transfer Unit C1.1.3
	        IF DB_ToteTracking.Transfer[_."B1.9.2"].toRight THEN
	            DB_ToteTracking.Conveyor[_."C1.3.1"].ToteDir.toLeft := FALSE;
	            DB_ToteTracking.Conveyor[_."C1.3.1"].ToteDir.toRight := TRUE;
	        END_IF;
	        // to Left for Transfer Unit C1.1.3
	        IF DB_ToteTracking.Transfer[_."B1.9.2"].toLeft THEN
	            DB_ToteTracking.Conveyor[_."C1.3.1"].ToteDir.toLeft := TRUE;
	            DB_ToteTracking.Conveyor[_."C1.3.1"].ToteDir.toRight := FALSE;
	        END_IF;
	        
	    END_REGION
	    
	END_REGION
	
	REGION C1.1.3 Right
	    
	    IF IDB_ProductionLine."B1.10.1".FilteredSensor AND
	        DB_ToteTracking.Conveyor[_."B1.10.1"].ToteDir.toRight AND
	        NOT IDB_ProductionLine."C1.3.1".ReadTransferStatus.Occupied
	    THEN
	        // Barcode
	        DB_ToteTracking.Conveyor[_."C1.3.1"].Barcode :=
	        DB_ToteTracking.Conveyor[_."B1.9.2"].Barcode;
	    END_IF;
	    
	END_REGION
	
	REGION B1.11.1 Straight
	    
	    IF IDB_ProductionLine."B1.10.1".FilteredSensor AND
	        DB_ToteTracking.Conveyor[_."B1.10.1"].ToteDir.Straight AND
	        NOT IDB_ProductionLine."B1.11.1".ReadConveyorStatus.Occupied
	    THEN
	        // Barcode
	        DB_ToteTracking.Conveyor[_."B1.11.1"].Barcode :=
	        DB_ToteTracking.Conveyor[_."B1.9.2"].Barcode;
	    END_IF;
	    
	END_REGION
	
	REGION C1.2.2
	    IF IDB_ProductionLine."C1.3.1".FilteredSensor AND
	        DB_ToteTracking.Conveyor[_."C1.3.1"].ToteDir.toRight AND
	        NOT IDB_ProductionLine."C1.2.2".ReadConveyorStatus.Occupied
	    THEN
	        DB_ToteTracking.Conveyor[_."C1.2.2"].Barcode :=
	        DB_ToteTracking.Conveyor[_."C1.3.1"].Barcode;
	    END_IF;
	    
	END_REGION
	
	REGION C1.4.1
	    IF IDB_ProductionLine."C1.3.1".FilteredSensor AND
	        DB_ToteTracking.Conveyor[_."C1.3.1"].ToteDir.toLeft  //AND
	        //NOT IDB_ProductionLine."C1.4.1".ReadConveyorStatus.Occupied
	    THEN
	        DB_ToteTracking.Conveyor[_."C1.4.1"].Barcode :=
	        DB_ToteTracking.Conveyor[_."C1.3.1"].Barcode;
	    END_IF;
	    
	END_REGION
	
	
	/////////////////////////////////////////////////////////
	//DP3
	////////////////////////////////////////////////////////
	
	REGION B1.17.1
	    
	    // write barcode data
	    DB_ToteTracking.Conveyor[_."B1.17.1"].Barcode :=
	    IDB_BarcodeReader.DP3.ResultStr;
	    
	END_REGION
	
	REGION B1.17.2
	    
	    IF IDB_ProductionLine."B1.17.1".CONVEYOR_SENSOR.SensorEdge.Negative THEN
	        // Barcode
	        DB_ToteTracking.Conveyor[_."B1.17.2"].Barcode :=
	        DB_ToteTracking.Conveyor[_."B1.17.1"].Barcode;
	        // main diverter direction
	        DB_ToteTracking.Conveyor[_."B1.17.2"].ToteDir :=
	        DB_ToteTracking.Conveyor[_."B1.17.1"].ToteDir;
	    END_IF;
	    
	END_REGION
	
	REGION B1.17.3
	    
	    IF IDB_ProductionLine."B1.17.2".CONVEYOR_SENSOR.SensorEdge.Negative THEN
	        // Barcode
	        DB_ToteTracking.Conveyor[_."B1.17.3"].Barcode :=
	        DB_ToteTracking.Conveyor[_."B1.17.2"].Barcode;
	        // main diverter direction
	        DB_ToteTracking.Conveyor[_."B1.17.3"].ToteDir :=
	        DB_ToteTracking.Conveyor[_."B1.17.2"].ToteDir;
	    END_IF;
	    
	END_REGION
	
	
	REGION B1.17.4
	    
	    IF IDB_ProductionLine."B1.17.3".CONVEYOR_SENSOR.SensorEdge.Negative
	    THEN
	        // Barcode
	        DB_ToteTracking.Conveyor[_."B1.17.4"].Barcode :=
	        DB_ToteTracking.Conveyor[_."B1.17.3"].Barcode;
	        // main diverter direction
	        DB_ToteTracking.Conveyor[_."B1.17.4"].ToteDir :=
	        DB_ToteTracking.Conveyor[_."B1.17.3"].ToteDir;
	    END_IF;
	    
	    
	    REGION Decision: Third diverter: before Transfer Unit 
	        
	        // to Left
	        IF DB_ToteTracking.Conveyor[_."B1.17.4"].ToteDir.toLeft OR
	           (DB_ToteTracking.Conveyor[_."B1.17.4"].Barcode = #NoReadTote) OR // bad read tote
	            _.Global.IDB_HardwareDiag."Cognex -10.106.129.24".CommunicationError // Cognex reader communcation error
	        THEN
	            DB_ToteTracking.Conveyor[_."B1.18.1"].ToteDir.Straight := FALSE;
	            DB_ToteTracking.Conveyor[_."B1.18.1"].ToteDir.toLeft := TRUE;
	        END_IF;
	        // to straight
	        IF DB_ToteTracking.Conveyor[_."B1.17.4"].ToteDir.Straight AND
	            NOT (DB_ToteTracking.Conveyor[_."B1.17.4"].Barcode = #NoReadTote) AND // Good read tote
	            NOT _.Global.IDB_HardwareDiag."Cognex -10.106.129.24".CommunicationError // Cognex reader communcation error
	        THEN
	            DB_ToteTracking.Conveyor[_."B1.18.1"].ToteDir.Straight := TRUE;
	            DB_ToteTracking.Conveyor[_."B1.18.1"].ToteDir.toLeft := FALSE;
	        END_IF;
	        
	    END_REGION
	    
	END_REGION
	
	REGION B1.6.1 Left
	    
	    IF IDB_ProductionLine."B1.18.1".FilteredSensor AND
	        DB_ToteTracking.Conveyor[_."B1.18.1"].ToteDir.toLeft AND
	        NOT IDB_S300_FullControl.ReadTransferStatus.Occupied
	    THEN
	        // Barcode
	        DB_ToteTracking.Conveyor[_."B1.6.1"].Barcode :=
	        DB_ToteTracking.Conveyor[_."B1.17.4"].Barcode;
	    END_IF;
	    
	END_REGION
	
	REGION B1.19.1 Straight
	    
	    IF IDB_ProductionLine."B1.18.1".FilteredSensor AND
	        DB_ToteTracking.Conveyor[_."B1.18.1"].ToteDir.Straight AND
	        NOT IDB_ProductionLine."B1.19.1".ReadConveyorStatus.Occupied
	    THEN
	        // Barcode
	        DB_ToteTracking.Conveyor[_."B1.19.1"].Barcode :=
	        DB_ToteTracking.Conveyor[_."B1.17.4"].Barcode;
	    END_IF;
	    
	END_REGION
	
	/////////////////////////////////////////////////////////
	//DP4
	////////////////////////////////////////////////////////
	
	REGION A1.7.4
	    
	    // write barcode data
	    DB_ToteTracking.Conveyor[_."A1.7.4"].Barcode :=
	    IDB_BarcodeReader.DP4.ResultStr;
	    
	END_REGION
	
	REGION A1.7.5
	    
	    IF IDB_ProductionLine."A1.7.4".CONVEYOR_SENSOR.SensorEdge.Negative THEN
	        // Barcode
	        DB_ToteTracking.Conveyor[_."A1.7.5"].Barcode :=
	        DB_ToteTracking.Conveyor[_."A1.7.4"].Barcode;
	        // main diverter direction
	        DB_ToteTracking.Conveyor[_."A1.7.5"].ToteDir :=
	        DB_ToteTracking.Conveyor[_."A1.7.4"].ToteDir;
	    END_IF;
	    
	END_REGION
	
	REGION A1.7.6
	    
	    IF IDB_ProductionLine."A1.7.5".CONVEYOR_SENSOR.SensorEdge.Negative THEN
	        // Barcode
	        DB_ToteTracking.Conveyor[_."A1.7.6"].Barcode :=
	        DB_ToteTracking.Conveyor[_."A1.7.5"].Barcode;
	        // main diverter direction
	        DB_ToteTracking.Conveyor[_."A1.7.6"].ToteDir :=
	        DB_ToteTracking.Conveyor[_."A1.7.5"].ToteDir;
	    END_IF;
	    
	END_REGION
	
	
	REGION A1.8.1
	    
	    IF IDB_ProductionLine."A1.7.6".CONVEYOR_SENSOR.SensorEdge.Negative
	    THEN
	        // Barcode
	        DB_ToteTracking.Conveyor[_."A1.8.1"].Barcode :=
	        DB_ToteTracking.Conveyor[_."A1.7.6"].Barcode;
	        // main diverter direction
	        DB_ToteTracking.Conveyor[_."A1.8.1"].ToteDir :=
	        DB_ToteTracking.Conveyor[_."A1.7.6"].ToteDir;
	    END_IF;
	    
	    
	    REGION Decision: main diverter: before Mabs
	        
	        // to Right
	        IF DB_ToteTracking.Conveyor[_."A1.8.1"].ToteDir.toRight OR
	            (DB_ToteTracking.Conveyor[_."A1.8.1"].Barcode = #NoReadTote) OR // bad read tote
	            _.Global.IDB_HardwareDiag."Cognex -10.106.129.24".CommunicationError // Cognex reader communcation error
	        THEN
	            DB_ToteTracking.Conveyor[_."A1.9.1"].ToteDir.Straight := FALSE;
	            DB_ToteTracking.Conveyor[_."A1.9.1"].ToteDir.toRight := TRUE;
	            DB_ToteTracking.Conveyor[_."A1.9.2"].ToteDir.Straight := FALSE;
	            DB_ToteTracking.Conveyor[_."A1.9.2"].ToteDir.toRight := TRUE;
	        END_IF;
	        // to straight
	        IF DB_ToteTracking.Conveyor[_."A1.8.1"].ToteDir.Straight AND
	            NOT (DB_ToteTracking.Conveyor[_."A1.8.1"].Barcode = #NoReadTote) AND // good read tote
	            NOT _.Global.IDB_HardwareDiag."Cognex -10.106.129.24".CommunicationError // Keyence reader communcation error
	        THEN
	            DB_ToteTracking.Conveyor[_."A1.9.1"].ToteDir.Straight := TRUE;
	            DB_ToteTracking.Conveyor[_."A1.9.1"].ToteDir.toRight := FALSE;
	            DB_ToteTracking.Conveyor[_."A1.9.2"].ToteDir.Straight := TRUE;
	            DB_ToteTracking.Conveyor[_."A1.9.2"].ToteDir.toRight := FALSE;
	        END_IF;
	        
	    END_REGION
	    
	END_REGION
	
	REGION D1.1.1 Right
	    
	    IF IDB_ProductionLine."A1.9.1".CROSS_SENSOR_FILTER.SensorEdge.Negative AND
	        NOT IDB_ProductionLine."A1.9.1".CurrentPosition.right AND  //remobve not
	        NOT IDB_ProductionLine."A1.9.2".CurrentPosition.right //AND  // remove not
	        //NOT IDB_ProductionLine."D1.1.1".ReadConveyorStatus.Occupied
	    THEN
	        // Barcode
	        DB_ToteTracking.Conveyor[_."D1.1.1"].Barcode :=
	        DB_ToteTracking.Conveyor[_."A1.8.1"].Barcode;
	    END_IF;
	    
	END_REGION
	
	REGION D1.1.2
	    
	    IF IDB_ProductionLine."D1.1.1".CONVEYOR_SENSOR.SensorEdge.Negative THEN
	        DB_ToteTracking.Conveyor[_."D1.2.1"] := DB_ToteTracking.Conveyor[_."D1.1.1"];
	    END_IF;
	    
	END_REGION
	
	REGION D1.2.1
	    
	    IF IDB_ProductionLine."D1.2.1".CONVEYOR_SENSOR.SensorEdge.Negative THEN
	        DB_ToteTracking.Conveyor[_."D1.3.1"] := DB_ToteTracking.Conveyor[_."D1.2.1"];
	    END_IF;
	    
	END_REGION
	
	
	REGION A1.10.1 Straight
	    
	    IF IDB_ProductionLine."A1.9.1".CROSS_SENSOR_FILTER.SensorEdge.Negative AND
	        NOT IDB_ProductionLine."A1.9.1".CurrentPosition.straight AND  //remove not
	        NOT IDB_ProductionLine."A1.9.2".CurrentPosition.straight //AND  // remove not
	        //NOT IDB_ProductionLine."A1.10.1".ReadConveyorStatus.Occupied
	    THEN
	        // Barcode
	        DB_ToteTracking.Conveyor[_."A1.10.1"].Barcode :=
	        DB_ToteTracking.Conveyor[_."A1.8.1"].Barcode;
	    END_IF;
	    
	END_REGION
	
	REGION A1.10.2
	    
	    IF IDB_ProductionLine."A1.10.1".CONVEYOR_SENSOR.SensorEdge.Negative THEN
	        DB_ToteTracking.Conveyor[_."A1.10.2"] := DB_ToteTracking.Conveyor[_."A1.10.1"];
	    END_IF;
	    
	END_REGION
	
	REGION A1.10.3
	    
	    IF IDB_ProductionLine."A1.10.2".CONVEYOR_SENSOR.SensorEdge.Negative THEN
	        DB_ToteTracking.Conveyor[_."A1.10.3"] := DB_ToteTracking.Conveyor[_."A1.10.2"];
	    END_IF;
	    
	END_REGION
	
	
	
	
END_FUNCTION_BLOCK
END_NAMESPACE

NAMESPACE Global
FUNCTION_BLOCK FB_StatusFault
{ S7_Optimized_Access := 'TRUE' ; Published := 'TRUE' }
VERSION : 0.1
   VAR_INPUT 
      FaultActive { ExternalAccessible := 'False'; ExternalVisible := 'False'; ExternalWritable := 'False'} : Bool;
      ResetFault { ExternalAccessible := 'False'; ExternalVisible := 'False'; ExternalWritable := 'False'} : Bool;
      StatusRunning : Bool;
      Feedback : Bool;
   END_VAR

   VAR_OUTPUT 
      FaultStatus { ExternalAccessible := 'False'; ExternalVisible := 'False'; ExternalWritable := 'False'} : Bool;
      FaultACK { ExternalAccessible := 'False'; ExternalVisible := 'False'; ExternalWritable := 'False'} : Bool;
   END_VAR

   VAR 
      FeedbackWatchdog {InstructionName := 'IEC_TIMER'; LibVersion := '1.0'; S7_SetPoint := 'False'} : IEC_TIMER;
      FeedbackError { S7_SetPoint := 'True'} : Bool;
      FeedbackTime : Time := T#1s;
      FeedbackLost : Bool;
   END_VAR


BEGIN
	// ==========================================================================================================================================================================
	// Company       : LogTech, s.r.o.
	// Created by    : Anton Vinoth Soundraraj
	// Block         : FB_StatusFault
	// Project       : LT-Lib-Block
	// ==========================================================================================================================================================================
	
	REGION Fault Status
	    
	    // init ack to 0
	    #FaultACK := 0;
	    
	    // ACTIVE --> FAULT STATUS
	    IF #FaultActive(* OR
	        #FeedbackError *)
	    THEN
	        #FaultStatus := TRUE;
	    END_IF;
	    
	    // RESET --> FAULT STATUS
	    IF #ResetFault AND
	        NOT #FaultActive
	    THEN
	        #FaultStatus := FALSE;
	        #FaultACK := TRUE;
	    END_IF;
	    
	    // Feedback watchdog check
	    
	    #FeedbackWatchdog.TON(IN:=#StatusRunning AND NOT #Feedback,
	                          PT:=#FeedbackTime,
	                          Q=>#FeedbackLost);
	    
	    // static to output
	    #FeedbackError :=
	    #FeedbackLost;
	    
	END_REGION
END_FUNCTION_BLOCK
END_NAMESPACE

NAMESPACE Global
FUNCTION_BLOCK FB_StatusReady
{ S7_Optimized_Access := 'TRUE' ; Published := 'TRUE' }
VERSION : 0.1
   VAR_INPUT 
      StatusON : Bool;
      StatusESTOP : Bool;
      StatusFAULT : Bool;
      StatusMAN : Bool;
      SignalFIRE : Bool;
      SystemAlertTime : Time;
   END_VAR

   VAR_OUTPUT 
      StatusReady : Bool;
   END_VAR

   VAR 
      StatusReadyCondition : Bool;
      SystemAlertTimer {InstructionName := 'IEC_TIMER'; LibVersion := '1.0'} : IEC_TIMER;
      SystemReadyToStart { S7_SetPoint := 'True'} : Bool;
   END_VAR


BEGIN
	// ==========================================================================================================================================================================
	// Company       : LogTech, s.r.o.
	// Created by    : Anton Vinoth Soundraraj
	// Block         : FB_StatusReady
	// Project       : LT-Lib-Block
	// ==========================================================================================================================================================================
	
	REGION Status Ready
	    
	    // Status ready condition
	    
	    #StatusReadyCondition :=
	    #StatusON AND
	    NOT #StatusESTOP AND
	    NOT #StatusFAULT AND
	    NOT #StatusMAN AND
	    NOT #SignalFIRE;
	    
	    #SystemAlertTimer.TON(IN := #StatusReadyCondition,
	                          PT := #SystemAlertTime,
	                          Q => #SystemReadyToStart);
	    
	    #StatusReady := #SystemReadyToStart;
	    
	END_REGION Status Ready
END_FUNCTION_BLOCK
END_NAMESPACE

NAMESPACE Global
FUNCTION_BLOCK FB_StatusON
{ S7_Optimized_Access := 'TRUE' ; Published := 'TRUE' }
VERSION : 0.1
   VAR_INPUT 
      SystemStartActive { ExternalAccessible := 'False'; ExternalVisible := 'False'; ExternalWritable := 'False'} : Bool;
      StatusStop { ExternalAccessible := 'False'; ExternalVisible := 'False'; ExternalWritable := 'False'} : Bool;
      StatusEStop { ExternalAccessible := 'False'; ExternalVisible := 'False'; ExternalWritable := 'False'} : Bool;
      StatusManual { ExternalAccessible := 'False'; ExternalVisible := 'False'; ExternalWritable := 'False'} : Bool;
      StatusFault { ExternalAccessible := 'False'; ExternalVisible := 'False'; ExternalWritable := 'False'} : Bool;
      FireAlarmActive { ExternalAccessible := 'False'; ExternalVisible := 'False'; ExternalWritable := 'False'} : Bool;
   END_VAR

   VAR_OUTPUT 
      StatusON { ExternalAccessible := 'False'; ExternalVisible := 'False'; ExternalWritable := 'False'} : Bool;
   END_VAR


BEGIN
	// ==========================================================================================================================================================================
	// Company       : LogTech, s.r.o.
	// Created by    : Anton Vinoth Soundraraj
	// Block         : FB_StatusON
	// Project       : LT-Lib-Block
	// ==========================================================================================================================================================================
	
	REGION STATUS ON
	    
	    IF #SystemStartActive AND NOT #StatusStop AND NOT #StatusEStop AND
	        NOT #StatusManual AND NOT #StatusFault AND NOT #FireAlarmActive
	    THEN
	        // The status of the conveyor is ON
	        #StatusON := TRUE;
	    END_IF;
	    
	    IF #StatusStop OR #StatusEStop OR #StatusManual OR
	        #StatusFault OR #FireAlarmActive THEN
	        // The status of the conveyor is OFF
	        #StatusON := FALSE;
	    END_IF;
	    
	END_REGION CONVEYOR STATUS ON
END_FUNCTION_BLOCK
END_NAMESPACE

DATA_BLOCK "FSIDB_Main_Safety_RTG1"   // DB1, F_DB
NAME : FUSI
// stored: InstanceOfName FSFB_Main_Safety_RTG1, InstanceOfType FB
"FSFB_Main_Safety_RTG1"
BEGIN
END_DATA_BLOCK

DATA_BLOCK "IDB_HardwareDiag"   // DB12
// stored: InstanceOfName Global.FB_HardwareDiag, InstanceOfType FB, Namespace Global
"Global.FB_HardwareDiag"
   // VAR
   //    ASi { S7_SetPoint := 'True'} : "LineA1.FB_GetDiag";
   // END_VAR
BEGIN
END_DATA_BLOCK

DATA_BLOCK "IDB_LineA1"   // DB8
// stored: InstanceOfName LineA1.FB_LineA1, InstanceOfType FB, Namespace LineA1
"LineA1.FB_LineA1"
   // VAR
   //    "Conveyor_A1.1.1" : "Global.FB_Conveyor";
   //    "MABS_A1.1.1" : "Global.FB_MABS";
   //    "Transfer_A1.1.1" : "Global.FB_S300_tTransMode";
   // END_VAR
BEGIN
END_DATA_BLOCK

DATA_BLOCK "IDB_LineB1"   // DB9
// stored: InstanceOfName LineB1.FB_LineB1, InstanceOfType FB, Namespace LineB1
"LineB1.FB_LineB1"
   // VAR
   //    "Conveyor_B1.1.1" : "Global.FB_Conveyor";
   //    "MABS_B1.1.1" : "Global.FB_MABS";
   //    "Transfer_B1.1.1" : "Global.FB_S300_tTransMode";
   //    "Transfer_B1.1.2" : "LineB1.FB_S300_FullControl";
   // END_VAR
BEGIN
END_DATA_BLOCK

